LIN {X 0,Y 573.287,Z 367.537,A -85,B 0,C 180,E1 -2259.17,E2 -2259.17} C_VEL
LIN {X 0,Y 573.427,Z 357.093,A -85,B 0,C 180,E1 -2260.058,E2 -2260.058} C_VEL
LIN {X 0,Y 573.544,Z 345.429,A -85,B 0,C 180,E1 -2260.853,E2 -2260.853} C_VEL
LIN {X 0,Y 573.652,Z 334.306,A -85,B 0,C 180,E1 -2261.446,E2 -2261.446} C_VEL
LIN {X 0,Y 573.759,Z 321.162,A -85,B 0,C 180,E1 -2261.974,E2 -2261.974} C_VEL
LIN {X 0,Y 573.832,Z 308.508,A -85,B 0,C 180,E1 -2262.332,E2 -2262.332} C_VEL
LIN {X 0,Y 573.943,Z 295.291,A -85,B 0,C 180,E1 -2262.554,E2 -2262.554} C_VEL
LIN {X 0,Y 573.968,Z 198.701,A -85,B 0,C 180,E1 -2263.769,E2 -2263.769} C_VEL
LIN {X 0,Y 573.396,Z 194.611,A -85,B 0,C 180,E1 -2263.851,E2 -2263.851} C_VEL
LIN {X 0,Y 573.568,Z 174.151,A -85,B 0,C 180,E1 -2266.723,E2 -2266.723} C_VEL
LIN {X 0,Y 573.787,Z 153.426,A -85,B 0,C 180,E1 -2269.647,E2 -2269.647} C_VEL
LIN {X 0,Y 573.932,Z 133.422,A -85,B 0,C 180,E1 -2272.499,E2 -2272.499} C_VEL
LIN {X 0,Y 573.536,Z 128.596,A -85,B 0,C 180,E1 -2273.214,E2 -2273.214} C_VEL
LIN {X 0,Y 573.23,Z 127.084,A -85,B 0,C 180,E1 -2273.466,E2 -2273.466} C_VEL
LIN {X 0,Y 573.214,Z 127.08,A -85,B 0,C 180,E1 -2276.487,E2 -2276.487} C_VEL
LIN {X 0,Y 573.242,Z 127.079,A -85,B 0,C 180,E1 -2279.367,E2 -2279.367} C_VEL
LIN {X 0,Y 573.24,Z 127.076,A -85,B 0,C 180,E1 -2282.226,E2 -2282.226} C_VEL
LIN {X 0,Y 573.225,Z 127.076,A -85,B 0,C 180,E1 -2284.769,E2 -2284.769} C_VEL
LIN {X 0,Y 573.23,Z 127.08,A -85,B 0,C 180,E1 -2287.808,E2 -2287.808} C_VEL
LIN {X 0,Y 573.25,Z 127.073,A -85,B 0,C 180,E1 -2290.525,E2 -2290.525} C_VEL
LIN {X 0,Y 573.21,Z 127.083,A -85,B 0,C 180,E1 -2293.665,E2 -2293.665} C_VEL
LIN {X 0,Y 573.205,Z 127.08,A -85,B 0,C 180,E1 -2296.637,E2 -2296.637} C_VEL
LIN {X 0,Y 573.251,Z 127.078,A -85,B 0,C 180,E1 -2299.475,E2 -2299.475} C_VEL
LIN {X 0,Y 573.23,Z 127.075,A -85,B 0,C 180,E1 -2302.192,E2 -2302.192} C_VEL
LIN {X 0,Y 573.227,Z 127.083,A -85,B 0,C 180,E1 -2305.231,E2 -2305.231} C_VEL
LIN {X 0,Y 573.242,Z 127.074,A -85,B 0,C 180,E1 -2307.774,E2 -2307.774} C_VEL
LIN {X 0,Y 573.236,Z 127.08,A -85,B 0,C 180,E1 -2310.632,E2 -2310.632} C_VEL
LIN {X 0,Y 573.217,Z 127.078,A -85,B 0,C 180,E1 -2313.513,E2 -2313.513} C_VEL
LIN {X 0,Y 573.197,Z 127.081,A -85,B 0,C 180,E1 -2316.133,E2 -2316.133} C_VEL
LIN {X 0,Y 573.232,Z 127.078,A -85,B 0,C 180,E1 -2319.172,E2 -2319.172} C_VEL
LIN {X 0,Y 573.199,Z 127.08,A -85,B 0,C 180,E1 -2321.41,E2 -2321.41} C_VEL
LIN {X 0,Y 573.208,Z 127.084,A -85,B 0,C 180,E1 -2324.351,E2 -2324.351} C_VEL
LIN {X 0,Y 573.196,Z 127.089,A -85,B 0,C 180,E1 -2326.528,E2 -2326.528} C_VEL
LIN {X 0,Y 573.261,Z 127.071,A -85,B 0,C 180,E1 -2329.403,E2 -2329.403} C_VEL
LIN {X 0,Y 573.245,Z 127.081,A -85,B 0,C 180,E1 -2332.249,E2 -2332.249} C_VEL
LIN {X 0,Y 573.279,Z 127.07,A -85,B 0,C 180,E1 -2335.077,E2 -2335.077} C_VEL
LIN {X 0,Y 573.31,Z 127.069,A -85,B 0,C 180,E1 -2337.892,E2 -2337.892} C_VEL
LIN {X 0,Y 573.32,Z 127.07,A -85,B 0,C 180,E1 -2339.999,E2 -2339.999} C_VEL
LIN {X 0,Y 573.277,Z 127.071,A -85,B 0,C 180,E1 -2342.81,E2 -2342.81} C_VEL
LIN {X 0,Y 573.269,Z 127.073,A -85,B 0,C 180,E1 -2345.628,E2 -2345.628} C_VEL
LIN {X 0,Y 573.238,Z 127.078,A -85,B 0,C 180,E1 -2348.46,E2 -2348.46} C_VEL
LIN {X 0,Y 573.239,Z 127.076,A -85,B 0,C 180,E1 -2351.312,E2 -2351.312} C_VEL
LIN {X 0,Y 573.245,Z 127.076,A -85,B 0,C 180,E1 -2354.408,E2 -2354.408} C_VEL
LIN {X 0,Y 573.178,Z 127.083,A -85,B 0,C 180,E1 -2357.113,E2 -2357.113} C_VEL
LIN {X 0,Y 573.206,Z 127.083,A -85,B 0,C 180,E1 -2360.078,E2 -2360.078} C_VEL
LIN {X 0,Y 573.197,Z 127.081,A -85,B 0,C 180,E1 -2362.339,E2 -2362.339} C_VEL
LIN {X 0,Y 573.195,Z 127.081,A -85,B 0,C 180,E1 -2364.348,E2 -2364.348} C_VEL
LIN {X 0,Y 572.558,Z 127.161,A -85,B 0,C 180,E1 -2364.934,E2 -2364.934} C_VEL
LIN {X 0,Y 569.726,Z 127.518,A -85,B 0,C 180,E1 -2365.886,E2 -2365.886} C_VEL
LIN {X 0,Y 567.304,Z 127.823,A -85,B 0,C 180,E1 -2366.652,E2 -2366.652} C_VEL
LIN {X 0,Y 566.246,Z 127.952,A -85,B 0,C 180,E1 -2367.243,E2 -2367.243} C_VEL
LIN {X 0,Y 566.151,Z 127.962,A -85,B 0,C 180,E1 -2367.443,E2 -2367.443} C_VEL
LIN {X 0,Y 566.148,Z 127.963,A -85,B 0,C 180,E1 -2369.771,E2 -2369.771} C_VEL
LIN {X 0,Y 566.19,Z 127.952,A -85,B 0,C 180,E1 -2372.427,E2 -2372.427} C_VEL
LIN {X 0,Y 566.162,Z 127.96,A -85,B 0,C 180,E1 -2374.986,E2 -2374.986} C_VEL
LIN {X 0,Y 566.186,Z 127.96,A -85,B 0,C 180,E1 -2377.461,E2 -2377.461} C_VEL
LIN {X 0,Y 566.192,Z 127.952,A -85,B 0,C 180,E1 -2380.199,E2 -2380.199} C_VEL
LIN {X 0,Y 566.174,Z 127.962,A -85,B 0,C 180,E1 -2383.056,E2 -2383.056} C_VEL
LIN {X 0,Y 566.152,Z 127.957,A -85,B 0,C 180,E1 -2386.053,E2 -2386.053} C_VEL
LIN {X 0,Y 566.15,Z 127.964,A -85,B 0,C 180,E1 -2388.858,E2 -2388.858} C_VEL
LIN {X 0,Y 566.197,Z 127.954,A -85,B 0,C 180,E1 -2391.442,E2 -2391.442} C_VEL
LIN {X 0,Y 566.134,Z 127.961,A -85,B 0,C 180,E1 -2394.305,E2 -2394.305} C_VEL
LIN {X 0,Y 566.187,Z 127.962,A -85,B 0,C 180,E1 -2396.895,E2 -2396.895} C_VEL
LIN {X 0,Y 566.152,Z 127.959,A -85,B 0,C 180,E1 -2399.405,E2 -2399.405} C_VEL
LIN {X 0,Y 566.141,Z 127.959,A -85,B 0,C 180,E1 -2401.853,E2 -2401.853} C_VEL
LIN {X 0,Y 566.18,Z 127.957,A -85,B 0,C 180,E1 -2404.249,E2 -2404.249} C_VEL
LIN {X 0,Y 566.149,Z 127.966,A -85,B 0,C 180,E1 -2406.722,E2 -2406.722} C_VEL
LIN {X 0,Y 566.182,Z 127.958,A -85,B 0,C 180,E1 -2408.901,E2 -2408.901} C_VEL
LIN {X 0,Y 566.175,Z 127.955,A -85,B 0,C 180,E1 -2411.171,E2 -2411.171} C_VEL
LIN {X 0,Y 566.16,Z 127.961,A -85,B 0,C 180,E1 -2414.151,E2 -2414.151} C_VEL
LIN {X 0,Y 566.154,Z 127.967,A -85,B 0,C 180,E1 -2416.358,E2 -2416.358} C_VEL
LIN {X 0,Y 566.202,Z 127.951,A -85,B 0,C 180,E1 -2419.269,E2 -2419.269} C_VEL
LIN {X 0,Y 566.18,Z 127.962,A -85,B 0,C 180,E1 -2422.152,E2 -2422.152} C_VEL
LIN {X 0,Y 566.242,Z 127.946,A -85,B 0,C 180,E1 -2425.016,E2 -2425.016} C_VEL
LIN {X 0,Y 566.272,Z 127.949,A -85,B 0,C 180,E1 -2427.866,E2 -2427.866} C_VEL
LIN {X 0,Y 566.278,Z 127.951,A -85,B 0,C 180,E1 -2430,E2 -2430} C_VEL
LIN {X 0,Y 566.205,Z 127.956,A -85,B 0,C 180,E1 -2432.846,E2 -2432.846} C_VEL
LIN {X 0,Y 566.349,Z 135.714,A -85,B 0,C 180,E1 -2434.27,E2 -2434.27} C_VEL
LIN {X 0,Y 566.262,Z 151.375,A -85,B 0,C 180,E1 -2437.129,E2 -2437.129} C_VEL
LIN {X 0,Y 566.198,Z 156.361,A -85,B 0,C 180,E1 -2438.042,E2 -2438.042} C_VEL
LIN {X 0,Y 567.178,Z 163.364,A -85,B 0,C 180,E1 -2438.167,E2 -2438.167} C_VEL
LIN {X 0,Y 566.934,Z 263.26,A -85,B 0,C 180,E1 -2439.454,E2 -2439.454} C_VEL
LIN {X 0,Y 566.794,Z 276.501,A -85,B 0,C 180,E1 -2439.771,E2 -2439.771} C_VEL
LIN {X 0,Y 566.723,Z 289.134,A -85,B 0,C 180,E1 -2440.224,E2 -2440.224} C_VEL
LIN {X 0,Y 566.591,Z 301.012,A -85,B 0,C 180,E1 -2440.801,E2 -2440.801} C_VEL
LIN {X 0,Y 566.411,Z 312.795,A -85,B 0,C 180,E1 -2441.541,E2 -2441.541} C_VEL
LIN {X 0,Y 566.309,Z 323.203,A -85,B 0,C 180,E1 -2442.361,E2 -2442.361} C_VEL
LIN {X 0,Y 566.179,Z 332.58,A -85,B 0,C 180,E1 -2443.276,E2 -2443.276} C_VEL
LIN {X 0,Y 566.081,Z 341.702,A -85,B 0,C 180,E1 -2444.377,E2 -2444.377} C_VEL
LIN {X 0,Y 566.009,Z 349.047,A -85,B 0,C 180,E1 -2445.483,E2 -2445.483} C_VEL
LIN {X 0,Y 565.939,Z 354.891,A -85,B 0,C 180,E1 -2446.596,E2 -2446.596} C_VEL
LIN {X 0,Y 565.918,Z 359.474,A -85,B 0,C 180,E1 -2447.714,E2 -2447.714} C_VEL
LIN {X 0,Y 565.872,Z 362.921,A -85,B 0,C 180,E1 -2448.839,E2 -2448.839} C_VEL
LIN {X 0,Y 565.841,Z 364.625,A -85,B 0,C 180,E1 -2449.594,E2 -2449.594} C_VEL
LIN {X 0,Y 565.856,Z 365.877,A -85,B 0,C 180,E1 -2450.351,E2 -2450.351} C_VEL
LIN {X 0,Y 565.87,Z 366.787,A -85,B 0,C 180,E1 -2451.335,E2 -2451.335} C_VEL
LIN {X 0,Y 565.838,Z 366.857,A -85,B 0,C 180,E1 -2452.646,E2 -2452.646} C_VEL
LIN {X 0,Y 565.844,Z 366.239,A -85,B 0,C 180,E1 -2453.419,E2 -2453.419} C_VEL
LIN {X 0,Y 565.828,Z 365.168,A -85,B 0,C 180,E1 -2454.198,E2 -2454.198} C_VEL
LIN {X 0,Y 565.908,Z 362.621,A -85,B 0,C 180,E1 -2455.37,E2 -2455.37} C_VEL
LIN {X 0,Y 565.965,Z 358.622,A -85,B 0,C 180,E1 -2456.612,E2 -2456.612} C_VEL
LIN {X 0,Y 565.944,Z 352.622,A -85,B 0,C 180,E1 -2457.956,E2 -2457.956} C_VEL
LIN {X 0,Y 566,Z 345.537,A -85,B 0,C 180,E1 -2459.168,E2 -2459.168} C_VEL
LIN {X 0,Y 566.115,Z 338.044,A -85,B 0,C 180,E1 -2460.184,E2 -2460.184} C_VEL
LIN {X 0,Y 566.242,Z 328.88,A -85,B 0,C 180,E1 -2461.196,E2 -2461.196} C_VEL
LIN {X 0,Y 566.325,Z 319.512,A -85,B 0,C 180,E1 -2462.041,E2 -2462.041} C_VEL
LIN {X 0,Y 566.452,Z 308.728,A -85,B 0,C 180,E1 -2462.826,E2 -2462.826} C_VEL
LIN {X 0,Y 566.637,Z 297.004,A -85,B 0,C 180,E1 -2463.5,E2 -2463.5} C_VEL
LIN {X 0,Y 566.77,Z 285.172,A -85,B 0,C 180,E1 -2464.025,E2 -2464.025} C_VEL
LIN {X 0,Y 566.859,Z 272.362,A -85,B 0,C 180,E1 -2464.435,E2 -2464.435} C_VEL
LIN {X 0,Y 566.968,Z 259.454,A -85,B 0,C 180,E1 -2464.697,E2 -2464.697} C_VEL
LIN {X 0,Y 567.051,Z 161.186,A -85,B 0,C 180,E1 -2465.954,E2 -2465.954} C_VEL
LIN {X 0,Y 566.24,Z 156.369,A -85,B 0,C 180,E1 -2466.045,E2 -2466.045} C_VEL
LIN {X 0,Y 566.424,Z 140.855,A -85,B 0,C 180,E1 -2468.883,E2 -2468.883} C_VEL
LIN {X 0,Y 566.44,Z 130.03,A -85,B 0,C 180,E1 -2470.814,E2 -2470.814} C_VEL
LIN {X 0,Y 566.25,Z 127.951,A -85,B 0,C 180,E1 -2471.222,E2 -2471.222} C_VEL
LIN {X 0,Y 566.197,Z 127.961,A -85,B 0,C 180,E1 -2474.036,E2 -2474.036} C_VEL
LIN {X 0,Y 566.202,Z 127.952,A -85,B 0,C 180,E1 -2477.083,E2 -2477.083} C_VEL
LIN {X 0,Y 566.224,Z 127.959,A -85,B 0,C 180,E1 -2479.803,E2 -2479.803} C_VEL
LIN {X 0,Y 566.196,Z 127.953,A -85,B 0,C 180,E1 -2482.6,E2 -2482.6} C_VEL
LIN {X 0,Y 566.197,Z 127.956,A -85,B 0,C 180,E1 -2485.182,E2 -2485.182} C_VEL
LIN {X 0,Y 566.23,Z 127.954,A -85,B 0,C 180,E1 -2487.744,E2 -2487.744} C_VEL
LIN {X 0,Y 566.202,Z 127.951,A -85,B 0,C 180,E1 -2490.329,E2 -2490.329} C_VEL
LIN {X 0,Y 566.211,Z 127.951,A -85,B 0,C 180,E1 -2492.662,E2 -2492.662} C_VEL
LIN {X 0,Y 566.236,Z 127.953,A -85,B 0,C 180,E1 -2495.04,E2 -2495.04} C_VEL
LIN {X 0,Y 566.193,Z 127.953,A -85,B 0,C 180,E1 -2498.138,E2 -2498.138} C_VEL
LIN {X 0,Y 566.231,Z 127.951,A -85,B 0,C 180,E1 -2500.615,E2 -2500.615} C_VEL
LIN {X 0,Y 566.201,Z 127.955,A -85,B 0,C 180,E1 -2503.413,E2 -2503.413} C_VEL
LIN {X 0,Y 566.186,Z 127.955,A -85,B 0,C 180,E1 -2506.359,E2 -2506.359} C_VEL
LIN {X 0,Y 566.237,Z 127.954,A -85,B 0,C 180,E1 -2508.676,E2 -2508.676} C_VEL
LIN {X 0,Y 566.205,Z 127.951,A -85,B 0,C 180,E1 -2511.435,E2 -2511.435} C_VEL
LIN {X 0,Y 566.263,Z 127.948,A -85,B 0,C 180,E1 -2514.302,E2 -2514.302} C_VEL
LIN {X 0,Y 566.282,Z 127.942,A -85,B 0,C 180,E1 -2517.867,E2 -2517.867} C_VEL
LIN {X 0,Y 566.297,Z 127.943,A -85,B 0,C 180,E1 -2520.712,E2 -2520.712} C_VEL
LIN {X 0,Y 566.255,Z 127.946,A -85,B 0,C 180,E1 -2522.846,E2 -2522.846} C_VEL
LIN {X 0,Y 566.25,Z 127.945,A -85,B 0,C 180,E1 -2525.699,E2 -2525.699} C_VEL
LIN {X 0,Y 566.2,Z 127.954,A -85,B 0,C 180,E1 -2528.567,E2 -2528.567} C_VEL
LIN {X 0,Y 566.243,Z 127.945,A -85,B 0,C 180,E1 -2531.455,E2 -2531.455} C_VEL
LIN {X 0,Y 566.222,Z 127.95,A -85,B 0,C 180,E1 -2534.5,E2 -2534.5} C_VEL
LIN {X 0,Y 566.154,Z 127.958,A -85,B 0,C 180,E1 -2537.334,E2 -2537.334} C_VEL
LIN {X 0,Y 566.194,Z 127.959,A -85,B 0,C 180,E1 -2539.582,E2 -2539.582} C_VEL
LIN {X 0,Y 566.15,Z 127.964,A -85,B 0,C 180,E1 -2541.865,E2 -2541.865} C_VEL
LIN {X 0,Y 566.182,Z 127.956,A -85,B 0,C 180,E1 -2545.021,E2 -2545.021} C_VEL
LIN {X 0,Y 566.16,Z 127.962,A -85,B 0,C 180,E1 -2547.342,E2 -2547.342} C_VEL
LIN {X 0,Y 566.148,Z 127.961,A -85,B 0,C 180,E1 -2549.772,E2 -2549.772} C_VEL
LIN {X 0,Y 566.173,Z 127.955,A -85,B 0,C 180,E1 -2552.425,E2 -2552.425} C_VEL
LIN {X 0,Y 566.152,Z 127.962,A -85,B 0,C 180,E1 -2554.985,E2 -2554.985} C_VEL
LIN {X 0,Y 566.178,Z 127.959,A -85,B 0,C 180,E1 -2557.463,E2 -2557.463} C_VEL
LIN {X 0,Y 566.162,Z 127.957,A -85,B 0,C 180,E1 -2560.203,E2 -2560.203} C_VEL
LIN {X 0,Y 566.148,Z 127.967,A -85,B 0,C 180,E1 -2563.06,E2 -2563.06} C_VEL
LIN {X 0,Y 566.157,Z 127.958,A -85,B 0,C 180,E1 -2566.054,E2 -2566.054} C_VEL
LIN {X 0,Y 566.163,Z 127.96,A -85,B 0,C 180,E1 -2569.22,E2 -2569.22} C_VEL
LIN {X 0,Y 566.173,Z 127.955,A -85,B 0,C 180,E1 -2571.636,E2 -2571.636} C_VEL
LIN {X 0,Y 566.141,Z 127.963,A -85,B 0,C 180,E1 -2574.306,E2 -2574.306} C_VEL
LIN {X 0,Y 566.196,Z 127.956,A -85,B 0,C 180,E1 -2576.896,E2 -2576.896} C_VEL
LIN {X 0,Y 566.169,Z 127.956,A -85,B 0,C 180,E1 -2579.406,E2 -2579.406} C_VEL
LIN {X 0,Y 566.151,Z 127.961,A -85,B 0,C 180,E1 -2581.854,E2 -2581.854} C_VEL
LIN {X 0,Y 566.194,Z 127.962,A -85,B 0,C 180,E1 -2584.25,E2 -2584.25} C_VEL
LIN {X 0,Y 566.203,Z 128.046,A -85,B 0,C 180,E1 -2586.451,E2 -2586.451} C_VEL
LIN {X 0,Y 566.985,Z 133.041,A -85,B 0,C 180,E1 -2587.21,E2 -2587.21} C_VEL
LIN {X 0,Y 566.812,Z 152.847,A -85,B 0,C 180,E1 -2590.064,E2 -2590.064} C_VEL
LIN {X 0,Y 566.588,Z 174.329,A -85,B 0,C 180,E1 -2593.112,E2 -2593.112} C_VEL
LIN {X 0,Y 566.39,Z 194.613,A -85,B 0,C 180,E1 -2595.975,E2 -2595.975} C_VEL
LIN {X 0,Y 567.155,Z 200.513,A -85,B 0,C 180,E1 -2596.085,E2 -2596.085} C_VEL
LIN {X 0,Y 566.961,Z 302.95,A -85,B 0,C 180,E1 -2597.403,E2 -2597.403} C_VEL
LIN {X 0,Y 566.84,Z 316.22,A -85,B 0,C 180,E1 -2597.719,E2 -2597.719} C_VEL
LIN {X 0,Y 566.743,Z 328.379,A -85,B 0,C 180,E1 -2598.148,E2 -2598.148} C_VEL
LIN {X 0,Y 566.604,Z 340.241,A -85,B 0,C 180,E1 -2598.713,E2 -2598.713} C_VEL
LIN {X 0,Y 566.439,Z 352.197,A -85,B 0,C 180,E1 -2599.455,E2 -2599.455} C_VEL
LIN {X 0,Y 566.325,Z 362.605,A -85,B 0,C 180,E1 -2600.266,E2 -2600.266} C_VEL
LIN {X 0,Y 566.207,Z 371.114,A -85,B 0,C 180,E1 -2601.074,E2 -2601.074} C_VEL
LIN {X 0,Y 566.112,Z 378.961,A -85,B 0,C 180,E1 -2601.972,E2 -2601.972} C_VEL
LIN {X 0,Y 566.004,Z 386.623,A -85,B 0,C 180,E1 -2603.047,E2 -2603.047} C_VEL
LIN {X 0,Y 566.004,Z 393.68,A -85,B 0,C 180,E1 -2604.299,E2 -2604.299} C_VEL
LIN {X 0,Y 565.933,Z 398.373,A -85,B 0,C 180,E1 -2605.37,E2 -2605.37} C_VEL
LIN {X 0,Y 565.927,Z 401.958,A -85,B 0,C 180,E1 -2606.44,E2 -2606.44} C_VEL
LIN {X 0,Y 565.878,Z 403.808,A -85,B 0,C 180,E1 -2607.153,E2 -2607.153} C_VEL
LIN {X 0,Y 565.846,Z 406.184,A -85,B 0,C 180,E1 -2608.577,E2 -2608.577} C_VEL
LIN {X 0,Y 565.839,Z 407,A -85,B 0,C 180,E1 -2610,E2 -2610} C_VEL
LIN {X 0,Y 565.846,Z 406.185,A -85,B 0,C 180,E1 -2611.424,E2 -2611.424} C_VEL
LIN {X 0,Y 565.878,Z 403.81,A -85,B 0,C 180,E1 -2612.848,E2 -2612.848} C_VEL
LIN {X 0,Y 565.926,Z 400.895,A -85,B 0,C 180,E1 -2613.917,E2 -2613.917} C_VEL
LIN {X 0,Y 565.878,Z 396.948,A -85,B 0,C 180,E1 -2614.988,E2 -2614.988} C_VEL
LIN {X 0,Y 566.002,Z 391.866,A -85,B 0,C 180,E1 -2616.059,E2 -2616.059} C_VEL
LIN {X 0,Y 566.041,Z 385.466,A -85,B 0,C 180,E1 -2617.132,E2 -2617.132} C_VEL
LIN {X 0,Y 566.134,Z 377.476,A -85,B 0,C 180,E1 -2618.208,E2 -2618.208} C_VEL
LIN {X 0,Y 566.229,Z 369.332,A -85,B 0,C 180,E1 -2619.106,E2 -2619.106} C_VEL
LIN {X 0,Y 566.348,Z 359.396,A -85,B 0,C 180,E1 -2620.005,E2 -2620.005} C_VEL
LIN {X 0,Y 566.536,Z 348.287,A -85,B 0,C 180,E1 -2620.807,E2 -2620.807} C_VEL
LIN {X 0,Y 566.614,Z 337.168,A -85,B 0,C 180,E1 -2621.447,E2 -2621.447} C_VEL
LIN {X 0,Y 566.746,Z 324.973,A -85,B 0,C 180,E1 -2621.988,E2 -2621.988} C_VEL
LIN {X 0,Y 566.914,Z 312.165,A -85,B 0,C 180,E1 -2622.394,E2 -2622.394} C_VEL
LIN {X 0,Y 566.991,Z 300.089,A -85,B 0,C 180,E1 -2622.642,E2 -2622.642} C_VEL
LIN {X 0,Y 567.089,Z 199.595,A -85,B 0,C 180,E1 -2623.928,E2 -2623.928} C_VEL
LIN {X 0,Y 566.392,Z 194.611,A -85,B 0,C 180,E1 -2624.026,E2 -2624.026} C_VEL
LIN {X 0,Y 566.589,Z 174.348,A -85,B 0,C 180,E1 -2626.889,E2 -2626.889} C_VEL
LIN {X 0,Y 566.864,Z 151.61,A -85,B 0,C 180,E1 -2630.124,E2 -2630.124} C_VEL
LIN {X 0,Y 567.001,Z 133.194,A -85,B 0,C 180,E1 -2632.79,E2 -2632.79} C_VEL
LIN {X 0,Y 566.198,Z 127.96,A -85,B 0,C 180,E1 -2633.598,E2 -2633.598} C_VEL
LIN {X 0,Y 566.19,Z 127.955,A -85,B 0,C 180,E1 -2636.543,E2 -2636.543} C_VEL
LIN {X 0,Y 566.173,Z 127.964,A -85,B 0,C 180,E1 -2639.771,E2 -2639.771} C_VEL
LIN {X 0,Y 566.196,Z 127.952,A -85,B 0,C 180,E1 -2642.428,E2 -2642.428} C_VEL
LIN {X 0,Y 566.17,Z 127.957,A -85,B 0,C 180,E1 -2644.987,E2 -2644.987} C_VEL
LIN {X 0,Y 566.194,Z 127.961,A -85,B 0,C 180,E1 -2647.461,E2 -2647.461} C_VEL
LIN {X 0,Y 566.209,Z 127.95,A -85,B 0,C 180,E1 -2650.199,E2 -2650.199} C_VEL
LIN {X 0,Y 566.183,Z 127.958,A -85,B 0,C 180,E1 -2653.056,E2 -2653.056} C_VEL
LIN {X 0,Y 566.16,Z 127.957,A -85,B 0,C 180,E1 -2656.053,E2 -2656.053} C_VEL
LIN {X 0,Y 566.168,Z 127.959,A -85,B 0,C 180,E1 -2658.859,E2 -2658.859} C_VEL
LIN {X 0,Y 566.207,Z 127.955,A -85,B 0,C 180,E1 -2661.443,E2 -2661.443} C_VEL
LIN {X 0,Y 566.146,Z 127.958,A -85,B 0,C 180,E1 -2664.306,E2 -2664.306} C_VEL
LIN {X 0,Y 566.199,Z 127.959,A -85,B 0,C 180,E1 -2666.896,E2 -2666.896} C_VEL
LIN {X 0,Y 566.164,Z 127.959,A -85,B 0,C 180,E1 -2669.406,E2 -2669.406} C_VEL
LIN {X 0,Y 566.154,Z 127.957,A -85,B 0,C 180,E1 -2671.854,E2 -2671.854} C_VEL
LIN {X 0,Y 566.192,Z 127.954,A -85,B 0,C 180,E1 -2674.249,E2 -2674.249} C_VEL
LIN {X 0,Y 566.144,Z 127.96,A -85,B 0,C 180,E1 -2677.366,E2 -2677.366} C_VEL
LIN {X 0,Y 566.174,Z 127.954,A -85,B 0,C 180,E1 -2679.661,E2 -2679.661} C_VEL
LIN {X 0,Y 566.169,Z 127.956,A -85,B 0,C 180,E1 -2681.92,E2 -2681.92} C_VEL
LIN {X 0,Y 566.183,Z 127.958,A -85,B 0,C 180,E1 -2684.89,E2 -2684.89} C_VEL
LIN {X 0,Y 566.177,Z 127.955,A -85,B 0,C 180,E1 -2687.817,E2 -2687.817} C_VEL
LIN {X 0,Y 566.17,Z 127.958,A -85,B 0,C 180,E1 -2689.991,E2 -2689.991} C_VEL
LIN {X 0,Y 566.192,Z 127.955,A -85,B 0,C 180,E1 -2692.869,E2 -2692.869} C_VEL
LIN {X 0,Y 566.255,Z 127.945,A -85,B 0,C 180,E1 -2695.015,E2 -2695.015} C_VEL
LIN {X 0,Y 566.28,Z 127.945,A -85,B 0,C 180,E1 -2697.866,E2 -2697.866} C_VEL
LIN {X 0,Y 566.289,Z 127.946,A -85,B 0,C 180,E1 -2699.999,E2 -2699.999} C_VEL
LIN {X 0,Y 566.245,Z 127.946,A -85,B 0,C 180,E1 -2702.845,E2 -2702.845} C_VEL
LIN {X 0,Y 566.238,Z 127.95,A -85,B 0,C 180,E1 -2705.698,E2 -2705.698} C_VEL
LIN {X 0,Y 566.19,Z 127.954,A -85,B 0,C 180,E1 -2708.566,E2 -2708.566} C_VEL
LIN {X 0,Y 566.197,Z 127.954,A -85,B 0,C 180,E1 -2711.455,E2 -2711.455} C_VEL
LIN {X 0,Y 566.206,Z 127.952,A -85,B 0,C 180,E1 -2714.493,E2 -2714.493} C_VEL
LIN {X 0,Y 566.152,Z 127.96,A -85,B 0,C 180,E1 -2717.332,E2 -2717.332} C_VEL
LIN {X 0,Y 566.176,Z 127.961,A -85,B 0,C 180,E1 -2719.581,E2 -2719.581} C_VEL
LIN {X 0,Y 566.149,Z 127.965,A -85,B 0,C 180,E1 -2721.864,E2 -2721.864} C_VEL
LIN {X 0,Y 566.195,Z 127.953,A -85,B 0,C 180,E1 -2724.962,E2 -2724.962} C_VEL
LIN {X 0,Y 566.151,Z 127.962,A -85,B 0,C 180,E1 -2727.443,E2 -2727.443} C_VEL
LIN {X 0,Y 565.456,Z 128.047,A -85,B 0,C 180,E1 -2728.037,E2 -2728.037} C_VEL
LIN {X 0,Y 562.581,Z 128.404,A -85,B 0,C 180,E1 -2729.001,E2 -2729.001} C_VEL
LIN {X 0,Y 560.182,Z 128.706,A -85,B 0,C 180,E1 -2729.776,E2 -2729.776} C_VEL
LIN {X 0,Y 559.172,Z 128.827,A -85,B 0,C 180,E1 -2730.375,E2 -2730.375} C_VEL
LIN {X 0,Y 559.101,Z 128.836,A -85,B 0,C 180,E1 -2730.578,E2 -2730.578} C_VEL
LIN {X 0,Y 559.146,Z 128.831,A -85,B 0,C 180,E1 -2732.715,E2 -2732.715} C_VEL
LIN {X 0,Y 559.113,Z 128.843,A -85,B 0,C 180,E1 -2735.324,E2 -2735.324} C_VEL
LIN {X 0,Y 559.12,Z 128.834,A -85,B 0,C 180,E1 -2738.018,E2 -2738.018} C_VEL
LIN {X 0,Y 559.146,Z 128.831,A -85,B 0,C 180,E1 -2739.939,E2 -2739.939} C_VEL
LIN {X 0,Y 559.12,Z 128.843,A -85,B 0,C 180,E1 -2743.193,E2 -2743.193} C_VEL
LIN {X 0,Y 559.119,Z 128.834,A -85,B 0,C 180,E1 -2745.763,E2 -2745.763} C_VEL
LIN {X 0,Y 559.097,Z 128.836,A -85,B 0,C 180,E1 -2748.223,E2 -2748.223} C_VEL
LIN {X 0,Y 559.164,Z 128.836,A -85,B 0,C 180,E1 -2751.065,E2 -2751.065} C_VEL
LIN {X 0,Y 559.111,Z 128.834,A -85,B 0,C 180,E1 -2753.787,E2 -2753.787} C_VEL
LIN {X 0,Y 559.138,Z 128.834,A -85,B 0,C 180,E1 -2756.423,E2 -2756.423} C_VEL
LIN {X 0,Y 559.135,Z 128.838,A -85,B 0,C 180,E1 -2758.979,E2 -2758.979} C_VEL
LIN {X 0,Y 559.102,Z 128.835,A -85,B 0,C 180,E1 -2761.63,E2 -2761.63} C_VEL
LIN {X 0,Y 559.147,Z 128.83,A -85,B 0,C 180,E1 -2763.901,E2 -2763.901} C_VEL
LIN {X 0,Y 559.097,Z 128.845,A -85,B 0,C 180,E1 -2766.58,E2 -2766.58} C_VEL
LIN {X 0,Y 559.14,Z 128.831,A -85,B 0,C 180,E1 -2769.394,E2 -2769.394} C_VEL
LIN {X 0,Y 559.106,Z 128.835,A -85,B 0,C 180,E1 -2771.684,E2 -2771.684} C_VEL
LIN {X 0,Y 559.119,Z 128.839,A -85,B 0,C 180,E1 -2774.694,E2 -2774.694} C_VEL
LIN {X 0,Y 559.137,Z 128.832,A -85,B 0,C 180,E1 -2777.662,E2 -2777.662} C_VEL
LIN {X 0,Y 559.111,Z 128.837,A -85,B 0,C 180,E1 -2779.864,E2 -2779.864} C_VEL
LIN {X 0,Y 559.14,Z 128.833,A -85,B 0,C 180,E1 -2782.779,E2 -2782.779} C_VEL
LIN {X 0,Y 559.219,Z 128.821,A -85,B 0,C 180,E1 -2784.953,E2 -2784.953} C_VEL
LIN {X 0,Y 559.242,Z 128.824,A -85,B 0,C 180,E1 -2787.839,E2 -2787.839} C_VEL
LIN {X 0,Y 559.246,Z 128.827,A -85,B 0,C 180,E1 -2790,E2 -2790} C_VEL
LIN {X 0,Y 559.207,Z 129.001,A -85,B 0,C 180,E1 -2792.791,E2 -2792.791} C_VEL
LIN {X 0,Y 559.333,Z 137.274,A -85,B 0,C 180,E1 -2794.323,E2 -2794.323} C_VEL
LIN {X 0,Y 559.255,Z 151.379,A -85,B 0,C 180,E1 -2796.901,E2 -2796.901} C_VEL
LIN {X 0,Y 559.205,Z 156.839,A -85,B 0,C 180,E1 -2797.878,E2 -2797.878} C_VEL
LIN {X 0,Y 560.298,Z 163.935,A -85,B 0,C 180,E1 -2797.999,E2 -2797.999} C_VEL
LIN {X 0,Y 560.014,Z 263.48,A -85,B 0,C 180,E1 -2799.298,E2 -2799.298} C_VEL
LIN {X 0,Y 559.859,Z 276.677,A -85,B 0,C 180,E1 -2799.62,E2 -2799.62} C_VEL
LIN {X 0,Y 559.761,Z 289.277,A -85,B 0,C 180,E1 -2800.078,E2 -2800.078} C_VEL
LIN {X 0,Y 559.617,Z 301.305,A -85,B 0,C 180,E1 -2800.675,E2 -2800.675} C_VEL
LIN {X 0,Y 559.421,Z 313.158,A -85,B 0,C 180,E1 -2801.435,E2 -2801.435} C_VEL
LIN {X 0,Y 559.295,Z 323.247,A -85,B 0,C 180,E1 -2802.242,E2 -2802.242} C_VEL
LIN {X 0,Y 559.144,Z 331.785,A -85,B 0,C 180,E1 -2803.076,E2 -2803.076} C_VEL
LIN {X 0,Y 559.032,Z 340.901,A -85,B 0,C 180,E1 -2804.172,E2 -2804.172} C_VEL
LIN {X 0,Y 558.925,Z 348.515,A -85,B 0,C 180,E1 -2805.311,E2 -2805.311} C_VEL
LIN {X 0,Y 558.858,Z 354.488,A -85,B 0,C 180,E1 -2806.436,E2 -2806.436} C_VEL
LIN {X 0,Y 558.83,Z 359.161,A -85,B 0,C 180,E1 -2807.568,E2 -2807.568} C_VEL
LIN {X 0,Y 558.787,Z 362.693,A -85,B 0,C 180,E1 -2808.706,E2 -2808.706} C_VEL
LIN {X 0,Y 558.743,Z 365.151,A -85,B 0,C 180,E1 -2809.853,E2 -2809.853} C_VEL
LIN {X 0,Y 558.761,Z 366.203,A -85,B 0,C 180,E1 -2810.621,E2 -2810.621} C_VEL
LIN {X 0,Y 558.762,Z 366.864,A -85,B 0,C 180,E1 -2811.449,E2 -2811.449} C_VEL
LIN {X 0,Y 558.737,Z 366.979,A -85,B 0,C 180,E1 -2812.17,E2 -2812.17} C_VEL
LIN {X 0,Y 558.754,Z 366.347,A -85,B 0,C 180,E1 -2813.339,E2 -2813.339} C_VEL
LIN {X 0,Y 558.76,Z 364.628,A -85,B 0,C 180,E1 -2814.524,E2 -2814.524} C_VEL
LIN {X 0,Y 558.817,Z 361.768,A -85,B 0,C 180,E1 -2815.715,E2 -2815.715} C_VEL
LIN {X 0,Y 558.841,Z 357.642,A -85,B 0,C 180,E1 -2816.919,E2 -2816.919} C_VEL
LIN {X 0,Y 558.882,Z 352.629,A -85,B 0,C 180,E1 -2818.029,E2 -2818.029} C_VEL
LIN {X 0,Y 558.924,Z 346.173,A -85,B 0,C 180,E1 -2819.16,E2 -2819.16} C_VEL
LIN {X 0,Y 559.053,Z 338.853,A -85,B 0,C 180,E1 -2820.189,E2 -2820.189} C_VEL
LIN {X 0,Y 559.183,Z 330.471,A -85,B 0,C 180,E1 -2821.15,E2 -2821.15} C_VEL
LIN {X 0,Y 559.302,Z 320.695,A -85,B 0,C 180,E1 -2822.066,E2 -2822.066} C_VEL
LIN {X 0,Y 559.446,Z 309.533,A -85,B 0,C 180,E1 -2822.91,E2 -2822.91} C_VEL
LIN {X 0,Y 559.668,Z 297.404,A -85,B 0,C 180,E1 -2823.625,E2 -2823.625} C_VEL
LIN {X 0,Y 559.831,Z 285.108,A -85,B 0,C 180,E1 -2824.181,E2 -2824.181} C_VEL
LIN {X 0,Y 559.935,Z 272.316,A -85,B 0,C 180,E1 -2824.594,E2 -2824.594} C_VEL
LIN {X 0,Y 560.07,Z 259.384,A -85,B 0,C 180,E1 -2824.858,E2 -2824.858} C_VEL
LIN {X 0,Y 560.25,Z 162.516,A -85,B 0,C 180,E1 -2826.111,E2 -2826.111} C_VEL
LIN {X 0,Y 559.214,Z 156.453,A -85,B 0,C 180,E1 -2826.235,E2 -2826.235} C_VEL
LIN {X 0,Y 559.431,Z 141.938,A -85,B 0,C 180,E1 -2828.913,E2 -2828.913} C_VEL
LIN {X 0,Y 559.332,Z 129.96,A -85,B 0,C 180,E1 -2831.072,E2 -2831.072} C_VEL
LIN {X 0,Y 559.196,Z 128.83,A -85,B 0,C 180,E1 -2831.296,E2 -2831.296} C_VEL
LIN {X 0,Y 559.152,Z 128.837,A -85,B 0,C 180,E1 -2834.24,E2 -2834.24} C_VEL
LIN {X 0,Y 559.161,Z 128.83,A -85,B 0,C 180,E1 -2837.258,E2 -2837.258} C_VEL
LIN {X 0,Y 559.183,Z 128.83,A -85,B 0,C 180,E1 -2840.136,E2 -2840.136} C_VEL
LIN {X 0,Y 559.138,Z 128.833,A -85,B 0,C 180,E1 -2842.892,E2 -2842.892} C_VEL
LIN {X 0,Y 559.164,Z 128.831,A -85,B 0,C 180,E1 -2846.052,E2 -2846.052} C_VEL
LIN {X 0,Y 559.154,Z 128.832,A -85,B 0,C 180,E1 -2848.981,E2 -2848.981} C_VEL
LIN {X 0,Y 559.167,Z 128.834,A -85,B 0,C 180,E1 -2851.62,E2 -2851.62} C_VEL
LIN {X 0,Y 559.179,Z 128.829,A -85,B 0,C 180,E1 -2853.904,E2 -2853.904} C_VEL
LIN {X 0,Y 559.141,Z 128.832,A -85,B 0,C 180,E1 -2856.572,E2 -2856.572} C_VEL
LIN {X 0,Y 559.175,Z 128.832,A -85,B 0,C 180,E1 -2859.396,E2 -2859.396} C_VEL
LIN {X 0,Y 559.133,Z 128.833,A -85,B 0,C 180,E1 -2861.686,E2 -2861.686} C_VEL
LIN {X 0,Y 559.156,Z 128.829,A -85,B 0,C 180,E1 -2863.948,E2 -2863.948} C_VEL
LIN {X 0,Y 559.16,Z 128.829,A -85,B 0,C 180,E1 -2866.184,E2 -2866.184} C_VEL
LIN {X 0,Y 559.208,Z 128.828,A -85,B 0,C 180,E1 -2868.605,E2 -2868.605} C_VEL
LIN {X 0,Y 559.169,Z 128.828,A -85,B 0,C 180,E1 -2871.326,E2 -2871.326} C_VEL
LIN {X 0,Y 559.231,Z 128.823,A -85,B 0,C 180,E1 -2874.23,E2 -2874.23} C_VEL
LIN {X 0,Y 559.253,Z 128.817,A -85,B 0,C 180,E1 -2877.84,E2 -2877.84} C_VEL
LIN {X 0,Y 559.268,Z 128.818,A -85,B 0,C 180,E1 -2880.721,E2 -2880.721} C_VEL
LIN {X 0,Y 559.222,Z 128.822,A -85,B 0,C 180,E1 -2882.882,E2 -2882.882} C_VEL
LIN {X 0,Y 559.219,Z 128.822,A -85,B 0,C 180,E1 -2885.771,E2 -2885.771} C_VEL
LIN {X 0,Y 559.165,Z 128.83,A -85,B 0,C 180,E1 -2888.675,E2 -2888.675} C_VEL
LIN {X 0,Y 559.204,Z 128.823,A -85,B 0,C 180,E1 -2891.601,E2 -2891.601} C_VEL
LIN {X 0,Y 559.185,Z 128.826,A -85,B 0,C 180,E1 -2894.588,E2 -2894.588} C_VEL
LIN {X 0,Y 559.112,Z 128.838,A -85,B 0,C 180,E1 -2897.559,E2 -2897.559} C_VEL
LIN {X 0,Y 559.148,Z 128.837,A -85,B 0,C 180,E1 -2899.839,E2 -2899.839} C_VEL
LIN {X 0,Y 559.105,Z 128.838,A -85,B 0,C 180,E1 -2902.155,E2 -2902.155} C_VEL
LIN {X 0,Y 559.142,Z 128.834,A -85,B 0,C 180,E1 -2905.178,E2 -2905.178} C_VEL
LIN {X 0,Y 559.102,Z 128.842,A -85,B 0,C 180,E1 -2907.717,E2 -2907.717} C_VEL
LIN {X 0,Y 559.094,Z 128.836,A -85,B 0,C 180,E1 -2910.187,E2 -2910.187} C_VEL
LIN {X 0,Y 559.135,Z 128.833,A -85,B 0,C 180,E1 -2912.717,E2 -2912.717} C_VEL
LIN {X 0,Y 559.109,Z 128.843,A -85,B 0,C 180,E1 -2915.326,E2 -2915.326} C_VEL
LIN {X 0,Y 559.098,Z 128.836,A -85,B 0,C 180,E1 -2918.021,E2 -2918.021} C_VEL
LIN {X 0,Y 559.099,Z 128.842,A -85,B 0,C 180,E1 -2920.818,E2 -2920.818} C_VEL
LIN {X 0,Y 559.101,Z 128.837,A -85,B 0,C 180,E1 -2923.738,E2 -2923.738} C_VEL
LIN {X 0,Y 559.102,Z 128.838,A -85,B 0,C 180,E1 -2926.262,E2 -2926.262} C_VEL
LIN {X 0,Y 559.116,Z 128.838,A -85,B 0,C 180,E1 -2929.184,E2 -2929.184} C_VEL
LIN {X 0,Y 559.168,Z 128.831,A -85,B 0,C 180,E1 -2931.193,E2 -2931.193} C_VEL
LIN {X 0,Y 559.118,Z 128.833,A -85,B 0,C 180,E1 -2933.788,E2 -2933.788} C_VEL
LIN {X 0,Y 559.147,Z 128.838,A -85,B 0,C 180,E1 -2936.424,E2 -2936.424} C_VEL
LIN {X 0,Y 559.15,Z 128.833,A -85,B 0,C 180,E1 -2938.98,E2 -2938.98} C_VEL
LIN {X 0,Y 559.112,Z 128.836,A -85,B 0,C 180,E1 -2941.63,E2 -2941.63} C_VEL
LIN {X 0,Y 559.159,Z 128.834,A -85,B 0,C 180,E1 -2943.902,E2 -2943.902} C_VEL
LIN {X 0,Y 559.163,Z 128.927,A -85,B 0,C 180,E1 -2946.311,E2 -2946.311} C_VEL
LIN {X 0,Y 560.048,Z 135.399,A -85,B 0,C 180,E1 -2947.302,E2 -2947.302} C_VEL
LIN {X 0,Y 559.797,Z 155.199,A -85,B 0,C 180,E1 -2950.186,E2 -2950.186} C_VEL
LIN {X 0,Y 559.568,Z 174.343,A -85,B 0,C 180,E1 -2952.936,E2 -2952.936} C_VEL
LIN {X 0,Y 559.374,Z 194.472,A -85,B 0,C 180,E1 -2955.795,E2 -2955.795} C_VEL
LIN {X 0,Y 560.255,Z 202.175,A -85,B 0,C 180,E1 -2955.934,E2 -2955.934} C_VEL
LIN {X 0,Y 560.033,Z 302.948,A -85,B 0,C 180,E1 -2957.245,E2 -2957.245} C_VEL
LIN {X 0,Y 559.913,Z 316.219,A -85,B 0,C 180,E1 -2957.564,E2 -2957.564} C_VEL
LIN {X 0,Y 559.792,Z 328.378,A -85,B 0,C 180,E1 -2957.999,E2 -2957.999} C_VEL
LIN {X 0,Y 559.644,Z 340.058,A -85,B 0,C 180,E1 -2958.56,E2 -2958.56} C_VEL
LIN {X 0,Y 559.458,Z 352.194,A -85,B 0,C 180,E1 -2959.322,E2 -2959.322} C_VEL
LIN {X 0,Y 559.305,Z 362.606,A -85,B 0,C 180,E1 -2960.142,E2 -2960.142} C_VEL
LIN {X 0,Y 559.162,Z 371.114,A -85,B 0,C 180,E1 -2960.961,E2 -2960.961} C_VEL
LIN {X 0,Y 559.05,Z 378.961,A -85,B 0,C 180,E1 -2961.87,E2 -2961.87} C_VEL
LIN {X 0,Y 558.944,Z 386.623,A -85,B 0,C 180,E1 -2962.958,E2 -2962.958} C_VEL
LIN {X 0,Y 558.936,Z 393.68,A -85,B 0,C 180,E1 -2964.227,E2 -2964.227} C_VEL
LIN {X 0,Y 558.826,Z 398.373,A -85,B 0,C 180,E1 -2965.311,E2 -2965.311} C_VEL
LIN {X 0,Y 558.836,Z 401.959,A -85,B 0,C 180,E1 -2966.395,E2 -2966.395} C_VEL
LIN {X 0,Y 558.799,Z 403.807,A -85,B 0,C 180,E1 -2967.116,E2 -2967.116} C_VEL
LIN {X 0,Y 558.745,Z 406.183,A -85,B 0,C 180,E1 -2968.559,E2 -2968.559} C_VEL
LIN {X 0,Y 558.74,Z 407,A -85,B 0,C 180,E1 -2970,E2 -2970} C_VEL
LIN {X 0,Y 558.745,Z 406.184,A -85,B 0,C 180,E1 -2971.442,E2 -2971.442} C_VEL
LIN {X 0,Y 558.799,Z 403.81,A -85,B 0,C 180,E1 -2972.884,E2 -2972.884} C_VEL
LIN {X 0,Y 558.844,Z 400.895,A -85,B 0,C 180,E1 -2973.966,E2 -2973.966} C_VEL
LIN {X 0,Y 558.798,Z 396.947,A -85,B 0,C 180,E1 -2975.051,E2 -2975.051} C_VEL
LIN {X 0,Y 558.922,Z 391.866,A -85,B 0,C 180,E1 -2976.136,E2 -2976.136} C_VEL
LIN {X 0,Y 558.978,Z 385.465,A -85,B 0,C 180,E1 -2977.223,E2 -2977.223} C_VEL
LIN {X 0,Y 559.099,Z 377.475,A -85,B 0,C 180,E1 -2978.312,E2 -2978.312} C_VEL
LIN {X 0,Y 559.195,Z 369.331,A -85,B 0,C 180,E1 -2979.221,E2 -2979.221} C_VEL
LIN {X 0,Y 559.358,Z 359.395,A -85,B 0,C 180,E1 -2980.131,E2 -2980.131} C_VEL
LIN {X 0,Y 559.556,Z 348.393,A -85,B 0,C 180,E1 -2980.937,E2 -2980.937} C_VEL
LIN {X 0,Y 559.673,Z 336.452,A -85,B 0,C 180,E1 -2981.628,E2 -2981.628} C_VEL
LIN {X 0,Y 559.822,Z 324.97,A -85,B 0,C 180,E1 -2982.139,E2 -2982.139} C_VEL
LIN {X 0,Y 559.979,Z 312.163,A -85,B 0,C 180,E1 -2982.55,E2 -2982.55} C_VEL
LIN {X 0,Y 560.08,Z 300.084,A -85,B 0,C 180,E1 -2982.801,E2 -2982.801} C_VEL
LIN {X 0,Y 560.201,Z 200.198,A -85,B 0,C 180,E1 -2984.093,E2 -2984.093} C_VEL
LIN {X 0,Y 559.373,Z 194.49,A -85,B 0,C 180,E1 -2984.205,E2 -2984.205} C_VEL
LIN {X 0,Y 559.57,Z 174.375,A -85,B 0,C 180,E1 -2987.069,E2 -2987.069} C_VEL
LIN {X 0,Y 559.888,Z 152.684,A -85,B 0,C 180,E1 -2990.194,E2 -2990.194} C_VEL
LIN {X 0,Y 560.057,Z 134.283,A -85,B 0,C 180,E1 -2992.893,E2 -2992.893} C_VEL
LIN {X 0,Y 559.156,Z 128.836,A -85,B 0,C 180,E1 -2993.766,E2 -2993.766} C_VEL
LIN {X 0,Y 559.127,Z 128.834,A -85,B 0,C 180,E1 -2996.818,E2 -2996.818} C_VEL
LIN {X 0,Y 559.123,Z 128.841,A -85,B 0,C 180,E1 -2999.852,E2 -2999.852} C_VEL
LIN {X 0,Y 559.151,Z 128.829,A -85,B 0,C 180,E1 -3002.716,E2 -3002.716} C_VEL
LIN {X 0,Y 559.121,Z 128.839,A -85,B 0,C 180,E1 -3005.325,E2 -3005.325} C_VEL
LIN {X 0,Y 559.13,Z 128.834,A -85,B 0,C 180,E1 -3008.018,E2 -3008.018} C_VEL
LIN {X 0,Y 559.157,Z 128.83,A -85,B 0,C 180,E1 -3010.813,E2 -3010.813} C_VEL
LIN {X 0,Y 559.111,Z 128.838,A -85,B 0,C 180,E1 -3013.737,E2 -3013.737} C_VEL
LIN {X 0,Y 559.111,Z 128.834,A -85,B 0,C 180,E1 -3016.263,E2 -3016.263} C_VEL
LIN {X 0,Y 559.157,Z 128.838,A -85,B 0,C 180,E1 -3019.187,E2 -3019.187} C_VEL
LIN {X 0,Y 559.131,Z 128.832,A -85,B 0,C 180,E1 -3021.982,E2 -3021.982} C_VEL
LIN {X 0,Y 559.127,Z 128.837,A -85,B 0,C 180,E1 -3024.789,E2 -3024.789} C_VEL
LIN {X 0,Y 559.153,Z 128.833,A -85,B 0,C 180,E1 -3027.366,E2 -3027.366} C_VEL
LIN {X 0,Y 559.114,Z 128.834,A -85,B 0,C 180,E1 -3030.15,E2 -3030.15} C_VEL
LIN {X 0,Y 559.13,Z 128.837,A -85,B 0,C 180,E1 -3033.182,E2 -3033.182} C_VEL
LIN {X 0,Y 559.11,Z 128.835,A -85,B 0,C 180,E1 -3035.492,E2 -3035.492} C_VEL
LIN {X 0,Y 559.164,Z 128.835,A -85,B 0,C 180,E1 -3038.623,E2 -3038.623} C_VEL
LIN {X 0,Y 559.16,Z 128.834,A -85,B 0,C 180,E1 -3040.925,E2 -3040.925} C_VEL
LIN {X 0,Y 559.13,Z 128.833,A -85,B 0,C 180,E1 -3043.946,E2 -3043.946} C_VEL
LIN {X 0,Y 559.139,Z 128.835,A -85,B 0,C 180,E1 -3046.183,E2 -3046.183} C_VEL
LIN {X 0,Y 559.195,Z 128.825,A -85,B 0,C 180,E1 -3049.133,E2 -3049.133} C_VEL
LIN {X 0,Y 559.181,Z 128.83,A -85,B 0,C 180,E1 -3052.053,E2 -3052.053} C_VEL
LIN {X 0,Y 559.232,Z 128.821,A -85,B 0,C 180,E1 -3054.953,E2 -3054.953} C_VEL
LIN {X 0,Y 559.251,Z 128.82,A -85,B 0,C 180,E1 -3057.839,E2 -3057.839} C_VEL
LIN {X 0,Y 559.258,Z 128.822,A -85,B 0,C 180,E1 -3059.999,E2 -3059.999} C_VEL
LIN {X 0,Y 559.213,Z 128.822,A -85,B 0,C 180,E1 -3062.881,E2 -3062.881} C_VEL
LIN {X 0,Y 559.207,Z 128.827,A -85,B 0,C 180,E1 -3065.77,E2 -3065.77} C_VEL
LIN {X 0,Y 559.155,Z 128.83,A -85,B 0,C 180,E1 -3068.674,E2 -3068.674} C_VEL
LIN {X 0,Y 559.159,Z 128.833,A -85,B 0,C 180,E1 -3071.601,E2 -3071.601} C_VEL
LIN {X 0,Y 559.155,Z 128.83,A -85,B 0,C 180,E1 -3074.575,E2 -3074.575} C_VEL
LIN {X 0,Y 559.111,Z 128.84,A -85,B 0,C 180,E1 -3077.558,E2 -3077.558} C_VEL
LIN {X 0,Y 559.139,Z 128.839,A -85,B 0,C 180,E1 -3079.838,E2 -3079.838} C_VEL
LIN {X 0,Y 559.104,Z 128.838,A -85,B 0,C 180,E1 -3082.154,E2 -3082.154} C_VEL
LIN {X 0,Y 559.14,Z 128.834,A -85,B 0,C 180,E1 -3085.177,E2 -3085.177} C_VEL
LIN {X 0,Y 559.101,Z 128.843,A -85,B 0,C 180,E1 -3087.716,E2 -3087.716} C_VEL
LIN {X 0,Y 559.101,Z 128.836,A -85,B 0,C 180,E1 -3090.578,E2 -3090.578} C_VEL
LIN {X 0,Y 558.461,Z 128.922,A -85,B 0,C 180,E1 -3091.18,E2 -3091.18} C_VEL
LIN {X 0,Y 555.612,Z 129.273,A -85,B 0,C 180,E1 -3092.156,E2 -3092.156} C_VEL
LIN {X 0,Y 553.194,Z 129.574,A -85,B 0,C 180,E1 -3092.942,E2 -3092.942} C_VEL
LIN {X 0,Y 552.162,Z 129.707,A -85,B 0,C 180,E1 -3093.549,E2 -3093.549} C_VEL
LIN {X 0,Y 552.083,Z 129.711,A -85,B 0,C 180,E1 -3093.754,E2 -3093.754} C_VEL
LIN {X 0,Y 552.095,Z 129.71,A -85,B 0,C 180,E1 -3096.747,E2 -3096.747} C_VEL
LIN {X 0,Y 552.119,Z 129.711,A -85,B 0,C 180,E1 -3099.527,E2 -3099.527} C_VEL
LIN {X 0,Y 552.08,Z 129.711,A -85,B 0,C 180,E1 -3102.429,E2 -3102.429} C_VEL
LIN {X 0,Y 552.07,Z 129.715,A -85,B 0,C 180,E1 -3105.559,E2 -3105.559} C_VEL
LIN {X 0,Y 552.056,Z 129.715,A -85,B 0,C 180,E1 -3108.548,E2 -3108.548} C_VEL
LIN {X 0,Y 552.107,Z 129.71,A -85,B 0,C 180,E1 -3111.41,E2 -3111.41} C_VEL
LIN {X 0,Y 552.064,Z 129.713,A -85,B 0,C 180,E1 -3114.154,E2 -3114.154} C_VEL
LIN {X 0,Y 552.1,Z 129.712,A -85,B 0,C 180,E1 -3117.155,E2 -3117.155} C_VEL
LIN {X 0,Y 552.071,Z 129.712,A -85,B 0,C 180,E1 -3119.956,E2 -3119.956} C_VEL
LIN {X 0,Y 552.084,Z 129.714,A -85,B 0,C 180,E1 -3123.009,E2 -3123.009} C_VEL
LIN {X 0,Y 552.067,Z 129.713,A -85,B 0,C 180,E1 -3125.96,E2 -3125.96} C_VEL
LIN {X 0,Y 552.088,Z 129.711,A -85,B 0,C 180,E1 -3129.118,E2 -3129.118} C_VEL
LIN {X 0,Y 552.069,Z 129.711,A -85,B 0,C 180,E1 -3131.442,E2 -3131.442} C_VEL
LIN {X 0,Y 552.077,Z 129.719,A -85,B 0,C 180,E1 -3134.494,E2 -3134.494} C_VEL
LIN {X 0,Y 552.09,Z 129.713,A -85,B 0,C 180,E1 -3136.754,E2 -3136.754} C_VEL
LIN {X 0,Y 552.076,Z 129.712,A -85,B 0,C 180,E1 -3139.734,E2 -3139.734} C_VEL
LIN {X 0,Y 552.1,Z 129.712,A -85,B 0,C 180,E1 -3141.95,E2 -3141.95} C_VEL
LIN {X 0,Y 552.196,Z 129.697,A -85,B 0,C 180,E1 -3144.888,E2 -3144.888} C_VEL
LIN {X 0,Y 552.213,Z 129.7,A -85,B 0,C 180,E1 -3147.812,E2 -3147.812} C_VEL
LIN {X 0,Y 552.215,Z 129.703,A -85,B 0,C 180,E1 -3150,E2 -3150} C_VEL
LIN {X 0,Y 552.184,Z 129.852,A -85,B 0,C 180,E1 -3152.69,E2 -3152.69} C_VEL
LIN {X 0,Y 552.336,Z 136.902,A -85,B 0,C 180,E1 -3154.013,E2 -3154.013} C_VEL
LIN {X 0,Y 552.268,Z 151.561,A -85,B 0,C 180,E1 -3156.704,E2 -3156.704} C_VEL
LIN {X 0,Y 552.189,Z 156.754,A -85,B 0,C 180,E1 -3157.678,E2 -3157.678} C_VEL
LIN {X 0,Y 553.42,Z 164.675,A -85,B 0,C 180,E1 -3157.827,E2 -3157.827} C_VEL
LIN {X 0,Y 553.09,Z 263.83,A -85,B 0,C 180,E1 -3159.139,E2 -3159.139} C_VEL
LIN {X 0,Y 552.928,Z 276.991,A -85,B 0,C 180,E1 -3159.465,E2 -3159.465} C_VEL
LIN {X 0,Y 552.816,Z 289.576,A -85,B 0,C 180,E1 -3159.929,E2 -3159.929} C_VEL
LIN {X 0,Y 552.653,Z 301.595,A -85,B 0,C 180,E1 -3160.533,E2 -3160.533} C_VEL
LIN {X 0,Y 552.442,Z 312.709,A -85,B 0,C 180,E1 -3161.251,E2 -3161.251} C_VEL
LIN {X 0,Y 552.301,Z 323.465,A -85,B 0,C 180,E1 -3162.12,E2 -3162.12} C_VEL
LIN {X 0,Y 552.111,Z 332.792,A -85,B 0,C 180,E1 -3163.058,E2 -3163.058} C_VEL
LIN {X 0,Y 551.978,Z 341.565,A -85,B 0,C 180,E1 -3164.148,E2 -3164.148} C_VEL
LIN {X 0,Y 551.857,Z 349.147,A -85,B 0,C 180,E1 -3165.323,E2 -3165.323} C_VEL
LIN {X 0,Y 551.782,Z 354.074,A -85,B 0,C 180,E1 -3166.273,E2 -3166.273} C_VEL
LIN {X 0,Y 551.744,Z 358.972,A -85,B 0,C 180,E1 -3167.455,E2 -3167.455} C_VEL
LIN {X 0,Y 551.697,Z 362.463,A -85,B 0,C 180,E1 -3168.57,E2 -3168.57} C_VEL
LIN {X 0,Y 551.676,Z 364.543,A -85,B 0,C 180,E1 -3169.491,E2 -3169.491} C_VEL
LIN {X 0,Y 551.655,Z 366.511,A -85,B 0,C 180,E1 -3170.899,E2 -3170.899} C_VEL
LIN {X 0,Y 551.645,Z 366.927,A -85,B 0,C 180,E1 -3171.682,E2 -3171.682} C_VEL
LIN {X 0,Y 551.64,Z 366.913,A -85,B 0,C 180,E1 -3172.47,E2 -3172.47} C_VEL
LIN {X 0,Y 551.654,Z 366.218,A -85,B 0,C 180,E1 -3173.472,E2 -3173.472} C_VEL
LIN {X 0,Y 551.682,Z 364.023,A -85,B 0,C 180,E1 -3174.859,E2 -3174.859} C_VEL
LIN {X 0,Y 551.74,Z 360.874,A -85,B 0,C 180,E1 -3176.069,E2 -3176.069} C_VEL
LIN {X 0,Y 551.773,Z 356.401,A -85,B 0,C 180,E1 -3177.293,E2 -3177.293} C_VEL
LIN {X 0,Y 551.829,Z 350.569,A -85,B 0,C 180,E1 -3178.507,E2 -3178.507} C_VEL
LIN {X 0,Y 551.899,Z 344.17,A -85,B 0,C 180,E1 -3179.568,E2 -3179.568} C_VEL
LIN {X 0,Y 552.026,Z 336.4,A -85,B 0,C 180,E1 -3180.614,E2 -3180.614} C_VEL
LIN {X 0,Y 552.213,Z 326.908,A -85,B 0,C 180,E1 -3181.646,E2 -3181.646} C_VEL
LIN {X 0,Y 552.38,Z 316.033,A -85,B 0,C 180,E1 -3182.592,E2 -3182.592} C_VEL
LIN {X 0,Y 552.612,Z 304.789,A -85,B 0,C 180,E1 -3183.37,E2 -3183.37} C_VEL
LIN {X 0,Y 552.782,Z 292.778,A -85,B 0,C 180,E1 -3184.015,E2 -3184.015} C_VEL
LIN {X 0,Y 552.941,Z 280.583,A -85,B 0,C 180,E1 -3184.509,E2 -3184.509} C_VEL
LIN {X 0,Y 553.071,Z 267.441,A -85,B 0,C 180,E1 -3184.878,E2 -3184.878} C_VEL
LIN {X 0,Y 553.131,Z 250.082,A -85,B 0,C 180,E1 -3185.151,E2 -3185.151} C_VEL
LIN {X 0,Y 553.302,Z 162.974,A -85,B 0,C 180,E1 -3186.288,E2 -3186.288} C_VEL
LIN {X 0,Y 552.198,Z 156.677,A -85,B 0,C 180,E1 -3186.405,E2 -3186.405} C_VEL
LIN {X 0,Y 552.432,Z 142.144,A -85,B 0,C 180,E1 -3189.102,E2 -3189.102} C_VEL
LIN {X 0,Y 552.344,Z 131.176,A -85,B 0,C 180,E1 -3191.102,E2 -3191.102} C_VEL
LIN {X 0,Y 552.188,Z 129.704,A -85,B 0,C 180,E1 -3191.396,E2 -3191.396} C_VEL
LIN {X 0,Y 552.093,Z 129.713,A -85,B 0,C 180,E1 -3194.533,E2 -3194.533} C_VEL
LIN {X 0,Y 552.128,Z 129.71,A -85,B 0,C 180,E1 -3197.585,E2 -3197.585} C_VEL
LIN {X 0,Y 552.132,Z 129.706,A -85,B 0,C 180,E1 -3200.474,E2 -3200.474} C_VEL
LIN {X 0,Y 552.104,Z 129.713,A -85,B 0,C 180,E1 -3203.318,E2 -3203.318} C_VEL
LIN {X 0,Y 552.125,Z 129.709,A -85,B 0,C 180,E1 -3205.94,E2 -3205.94} C_VEL
LIN {X 0,Y 552.117,Z 129.706,A -85,B 0,C 180,E1 -3208.541,E2 -3208.541} C_VEL
LIN {X 0,Y 552.123,Z 129.715,A -85,B 0,C 180,E1 -3211.439,E2 -3211.439} C_VEL
LIN {X 0,Y 552.129,Z 129.705,A -85,B 0,C 180,E1 -3214.357,E2 -3214.357} C_VEL
LIN {X 0,Y 552.098,Z 129.711,A -85,B 0,C 180,E1 -3216.759,E2 -3216.759} C_VEL
LIN {X 0,Y 552.118,Z 129.714,A -85,B 0,C 180,E1 -3219.12,E2 -3219.12} C_VEL
LIN {X 0,Y 552.091,Z 129.713,A -85,B 0,C 180,E1 -3221.444,E2 -3221.444} C_VEL
LIN {X 0,Y 552.105,Z 129.708,A -85,B 0,C 180,E1 -3223.738,E2 -3223.738} C_VEL
LIN {X 0,Y 552.123,Z 129.705,A -85,B 0,C 180,E1 -3226.005,E2 -3226.005} C_VEL
LIN {X 0,Y 552.162,Z 129.707,A -85,B 0,C 180,E1 -3228.994,E2 -3228.994} C_VEL
LIN {X 0,Y 552.151,Z 129.701,A -85,B 0,C 180,E1 -3231.952,E2 -3231.952} C_VEL
LIN {X 0,Y 552.222,Z 129.696,A -85,B 0,C 180,E1 -3234.89,E2 -3234.89} C_VEL
LIN {X 0,Y 552.224,Z 129.693,A -85,B 0,C 180,E1 -3237.813,E2 -3237.813} C_VEL
LIN {X 0,Y 552.238,Z 129.693,A -85,B 0,C 180,E1 -3240.73,E2 -3240.73} C_VEL
LIN {X 0,Y 552.188,Z 129.698,A -85,B 0,C 180,E1 -3242.919,E2 -3242.919} C_VEL
LIN {X 0,Y 552.188,Z 129.698,A -85,B 0,C 180,E1 -3245.845,E2 -3245.845} C_VEL
LIN {X 0,Y 552.136,Z 129.704,A -85,B 0,C 180,E1 -3248.787,E2 -3248.787} C_VEL
LIN {X 0,Y 552.16,Z 129.702,A -85,B 0,C 180,E1 -3251.751,E2 -3251.751} C_VEL
LIN {X 0,Y 552.131,Z 129.704,A -85,B 0,C 180,E1 -3254.749,E2 -3254.749} C_VEL
LIN {X 0,Y 552.078,Z 129.718,A -85,B 0,C 180,E1 -3257.79,E2 -3257.79} C_VEL
LIN {X 0,Y 552.1,Z 129.711,A -85,B 0,C 180,E1 -3260.103,E2 -3260.103} C_VEL
LIN {X 0,Y 552.045,Z 129.715,A -85,B 0,C 180,E1 -3262.454,E2 -3262.454} C_VEL
LIN {X 0,Y 552.085,Z 129.715,A -85,B 0,C 180,E1 -3265.334,E2 -3265.334} C_VEL
LIN {X 0,Y 552.05,Z 129.716,A -85,B 0,C 180,E1 -3268.102,E2 -3268.102} C_VEL
LIN {X 0,Y 552.069,Z 129.711,A -85,B 0,C 180,E1 -3270.612,E2 -3270.612} C_VEL
LIN {X 0,Y 552.09,Z 129.717,A -85,B 0,C 180,E1 -3273.188,E2 -3273.188} C_VEL
LIN {X 0,Y 552.064,Z 129.714,A -85,B 0,C 180,E1 -3275.846,E2 -3275.846} C_VEL
LIN {X 0,Y 552.074,Z 129.713,A -85,B 0,C 180,E1 -3278.593,E2 -3278.593} C_VEL
LIN {X 0,Y 552.055,Z 129.718,A -85,B 0,C 180,E1 -3281.453,E2 -3281.453} C_VEL
LIN {X 0,Y 552.076,Z 129.715,A -85,B 0,C 180,E1 -3284.53,E2 -3284.53} C_VEL
LIN {X 0,Y 552.082,Z 129.712,A -85,B 0,C 180,E1 -3287.591,E2 -3287.591} C_VEL
LIN {X 0,Y 552.123,Z 129.712,A -85,B 0,C 180,E1 -3290.472,E2 -3290.472} C_VEL
LIN {X 0,Y 552.099,Z 129.708,A -85,B 0,C 180,E1 -3293.319,E2 -3293.319} C_VEL
LIN {X 0,Y 552.099,Z 129.71,A -85,B 0,C 180,E1 -3295.937,E2 -3295.937} C_VEL
LIN {X 0,Y 552.123,Z 129.714,A -85,B 0,C 180,E1 -3298.541,E2 -3298.541} C_VEL
LIN {X 0,Y 552.081,Z 129.712,A -85,B 0,C 180,E1 -3301.447,E2 -3301.447} C_VEL
LIN {X 0,Y 552.085,Z 129.719,A -85,B 0,C 180,E1 -3304.354,E2 -3304.354} C_VEL
LIN {X 0,Y 552.132,Z 129.908,A -85,B 0,C 180,E1 -3306.183,E2 -3306.183} C_VEL
LIN {X 0,Y 553.094,Z 136.433,A -85,B 0,C 180,E1 -3307.198,E2 -3307.198} C_VEL
LIN {X 0,Y 552.852,Z 154.917,A -85,B 0,C 180,E1 -3309.926,E2 -3309.926} C_VEL
LIN {X 0,Y 552.559,Z 174.836,A -85,B 0,C 180,E1 -3312.824,E2 -3312.824} C_VEL
LIN {X 0,Y 552.362,Z 194.31,A -85,B 0,C 180,E1 -3315.627,E2 -3315.627} C_VEL
LIN {X 0,Y 553.357,Z 202.397,A -85,B 0,C 180,E1 -3315.762,E2 -3315.762} C_VEL
LIN {X 0,Y 553.104,Z 302.624,A -85,B 0,C 180,E1 -3317.082,E2 -3317.082} C_VEL
LIN {X 0,Y 552.98,Z 315.938,A -85,B 0,C 180,E1 -3317.406,E2 -3317.406} C_VEL
LIN {X 0,Y 552.847,Z 328.133,A -85,B 0,C 180,E1 -3317.846,E2 -3317.846} C_VEL
LIN {X 0,Y 552.657,Z 338.966,A -85,B 0,C 180,E1 -3318.365,E2 -3318.365} C_VEL
LIN {X 0,Y 552.482,Z 350.76,A -85,B 0,C 180,E1 -3319.093,E2 -3319.093} C_VEL
LIN {X 0,Y 552.298,Z 361.448,A -85,B 0,C 180,E1 -3319.923,E2 -3319.923} C_VEL
LIN {X 0,Y 552.131,Z 371.079,A -85,B 0,C 180,E1 -3320.845,E2 -3320.845} C_VEL
LIN {X 0,Y 552.013,Z 378.961,A -85,B 0,C 180,E1 -3321.765,E2 -3321.765} C_VEL
LIN {X 0,Y 551.89,Z 386.622,A -85,B 0,C 180,E1 -3322.868,E2 -3322.868} C_VEL
LIN {X 0,Y 551.867,Z 393.68,A -85,B 0,C 180,E1 -3324.153,E2 -3324.153} C_VEL
LIN {X 0,Y 551.725,Z 398.373,A -85,B 0,C 180,E1 -3325.251,E2 -3325.251} C_VEL
LIN {X 0,Y 551.75,Z 401.958,A -85,B 0,C 180,E1 -3326.349,E2 -3326.349} C_VEL
LIN {X 0,Y 551.724,Z 403.807,A -85,B 0,C 180,E1 -3327.079,E2 -3327.079} C_VEL
LIN {X 0,Y 551.645,Z 406.182,A -85,B 0,C 180,E1 -3328.54,E2 -3328.54} C_VEL
LIN {X 0,Y 551.64,Z 407,A -85,B 0,C 180,E1 -3330,E2 -3330} C_VEL
LIN {X 0,Y 551.645,Z 406.183,A -85,B 0,C 180,E1 -3331.46,E2 -3331.46} C_VEL
LIN {X 0,Y 551.724,Z 403.81,A -85,B 0,C 180,E1 -3332.921,E2 -3332.921} C_VEL
LIN {X 0,Y 551.764,Z 400.895,A -85,B 0,C 180,E1 -3334.017,E2 -3334.017} C_VEL
LIN {X 0,Y 551.724,Z 396.947,A -85,B 0,C 180,E1 -3335.116,E2 -3335.116} C_VEL
LIN {X 0,Y 551.825,Z 391.191,A -85,B 0,C 180,E1 -3336.341,E2 -3336.341} C_VEL
LIN {X 0,Y 551.927,Z 384.234,A -85,B 0,C 180,E1 -3337.5,E2 -3337.5} C_VEL
LIN {X 0,Y 552.083,Z 375.985,A -85,B 0,C 180,E1 -3338.603,E2 -3338.603} C_VEL
LIN {X 0,Y 552.201,Z 367.485,A -85,B 0,C 180,E1 -3339.524,E2 -3339.524} C_VEL
LIN {X 0,Y 552.429,Z 356.983,A -85,B 0,C 180,E1 -3340.445,E2 -3340.445} C_VEL
LIN {X 0,Y 552.576,Z 346.127,A -85,B 0,C 180,E1 -3341.214,E2 -3341.214} C_VEL
LIN {X 0,Y 552.753,Z 335.201,A -85,B 0,C 180,E1 -3341.831,E2 -3341.831} C_VEL
LIN {X 0,Y 552.899,Z 323.515,A -85,B 0,C 180,E1 -3342.34,E2 -3342.34} C_VEL
LIN {X 0,Y 553.037,Z 310.966,A -85,B 0,C 180,E1 -3342.733,E2 -3342.733} C_VEL
LIN {X 0,Y 553.204,Z 298.257,A -85,B 0,C 180,E1 -3342.986,E2 -3342.986} C_VEL
LIN {X 0,Y 553.233,Z 200.351,A -85,B 0,C 180,E1 -3344.269,E2 -3344.269} C_VEL
LIN {X 0,Y 552.346,Z 194.229,A -85,B 0,C 180,E1 -3344.393,E2 -3344.393} C_VEL
LIN {X 0,Y 552.583,Z 173.738,A -85,B 0,C 180,E1 -3347.35,E2 -3347.35} C_VEL
LIN {X 0,Y 552.941,Z 152.444,A -85,B 0,C 180,E1 -3350.459,E2 -3350.459} C_VEL
LIN {X 0,Y 553.083,Z 135.372,A -85,B 0,C 180,E1 -3353.001,E2 -3353.001} C_VEL
LIN {X 0,Y 552.085,Z 129.716,A -85,B 0,C 180,E1 -3353.916,E2 -3353.916} C_VEL
LIN {X 0,Y 552.096,Z 129.711,A -85,B 0,C 180,E1 -3356.99,E2 -3356.99} C_VEL
LIN {X 0,Y 552.099,Z 129.713,A -85,B 0,C 180,E1 -3360.047,E2 -3360.047} C_VEL
LIN {X 0,Y 552.111,Z 129.707,A -85,B 0,C 180,E1 -3362.845,E2 -3362.845} C_VEL
LIN {X 0,Y 552.075,Z 129.715,A -85,B 0,C 180,E1 -3365.845,E2 -3365.845} C_VEL
LIN {X 0,Y 552.116,Z 129.706,A -85,B 0,C 180,E1 -3368.59,E2 -3368.59} C_VEL
LIN {X 0,Y 552.078,Z 129.719,A -85,B 0,C 180,E1 -3371.45,E2 -3371.45} C_VEL
LIN {X 0,Y 552.079,Z 129.711,A -85,B 0,C 180,E1 -3374.529,E2 -3374.529} C_VEL
LIN {X 0,Y 552.091,Z 129.713,A -85,B 0,C 180,E1 -3377.59,E2 -3377.59} C_VEL
LIN {X 0,Y 552.13,Z 129.705,A -85,B 0,C 180,E1 -3380.472,E2 -3380.472} C_VEL
LIN {X 0,Y 552.103,Z 129.713,A -85,B 0,C 180,E1 -3383.318,E2 -3383.318} C_VEL
LIN {X 0,Y 552.102,Z 129.707,A -85,B 0,C 180,E1 -3385.937,E2 -3385.937} C_VEL
LIN {X 0,Y 552.084,Z 129.713,A -85,B 0,C 180,E1 -3388.538,E2 -3388.538} C_VEL
LIN {X 0,Y 552.083,Z 129.712,A -85,B 0,C 180,E1 -3391.447,E2 -3391.447} C_VEL
LIN {X 0,Y 552.087,Z 129.712,A -85,B 0,C 180,E1 -3394.353,E2 -3394.353} C_VEL
LIN {X 0,Y 552.072,Z 129.72,A -85,B 0,C 180,E1 -3396.756,E2 -3396.756} C_VEL
LIN {X 0,Y 552.101,Z 129.711,A -85,B 0,C 180,E1 -3399.119,E2 -3399.119} C_VEL
LIN {X 0,Y 552.083,Z 129.71,A -85,B 0,C 180,E1 -3401.442,E2 -3401.442} C_VEL
LIN {X 0,Y 552.09,Z 129.717,A -85,B 0,C 180,E1 -3404.494,E2 -3404.494} C_VEL
LIN {X 0,Y 552.107,Z 129.707,A -85,B 0,C 180,E1 -3407.502,E2 -3407.502} C_VEL
LIN {X 0,Y 552.1,Z 129.708,A -85,B 0,C 180,E1 -3409.734,E2 -3409.734} C_VEL
LIN {X 0,Y 552.139,Z 129.706,A -85,B 0,C 180,E1 -3411.951,E2 -3411.951} C_VEL
LIN {X 0,Y 552.209,Z 129.696,A -85,B 0,C 180,E1 -3414.888,E2 -3414.888} C_VEL
LIN {X 0,Y 552.222,Z 129.695,A -85,B 0,C 180,E1 -3417.811,E2 -3417.811} C_VEL
LIN {X 0,Y 552.226,Z 129.698,A -85,B 0,C 180,E1 -3419.999,E2 -3419.999} C_VEL
LIN {X 0,Y 552.18,Z 129.698,A -85,B 0,C 180,E1 -3422.918,E2 -3422.918} C_VEL
LIN {X 0,Y 552.177,Z 129.704,A -85,B 0,C 180,E1 -3425.843,E2 -3425.843} C_VEL
LIN {X 0,Y 552.127,Z 129.705,A -85,B 0,C 180,E1 -3428.786,E2 -3428.786} C_VEL
LIN {X 0,Y 552.105,Z 129.713,A -85,B 0,C 180,E1 -3431.751,E2 -3431.751} C_VEL
LIN {X 0,Y 552.122,Z 129.705,A -85,B 0,C 180,E1 -3434.748,E2 -3434.748} C_VEL
LIN {X 0,Y 552.075,Z 129.721,A -85,B 0,C 180,E1 -3437.789,E2 -3437.789} C_VEL
LIN {X 0,Y 552.094,Z 129.712,A -85,B 0,C 180,E1 -3440.102,E2 -3440.102} C_VEL
LIN {X 0,Y 552.045,Z 129.715,A -85,B 0,C 180,E1 -3442.452,E2 -3442.452} C_VEL
LIN {X 0,Y 552.083,Z 129.715,A -85,B 0,C 180,E1 -3445.333,E2 -3445.333} C_VEL
LIN {X 0,Y 552.049,Z 129.716,A -85,B 0,C 180,E1 -3448.101,E2 -3448.101} C_VEL
LIN {X 0,Y 552.07,Z 129.711,A -85,B 0,C 180,E1 -3450.61,E2 -3450.61} C_VEL
LIN {X 0,Y 552.102,Z 129.713,A -85,B 0,C 180,E1 -3453.186,E2 -3453.186} C_VEL
LIN {X 0,Y 552.083,Z 129.711,A -85,B 0,C 180,E1 -3453.754,E2 -3453.754} C_VEL
LIN {X 0,Y 551.44,Z 129.793,A -85,B 0,C 180,E1 -3454.363,E2 -3454.363} C_VEL
LIN {X 0,Y 548.629,Z 130.149,A -85,B 0,C 180,E1 -3455.351,E2 -3455.351} C_VEL
LIN {X 0,Y 546.223,Z 130.444,A -85,B 0,C 180,E1 -3456.147,E2 -3456.147} C_VEL
LIN {X 0,Y 545.159,Z 130.574,A -85,B 0,C 180,E1 -3456.761,E2 -3456.761} C_VEL
LIN {X 0,Y 545.056,Z 130.589,A -85,B 0,C 180,E1 -3456.969,E2 -3456.969} C_VEL
LIN {X 0,Y 545.048,Z 130.586,A -85,B 0,C 180,E1 -3460.143,E2 -3460.143} C_VEL
LIN {X 0,Y 545.013,Z 130.599,A -85,B 0,C 180,E1 -3463.112,E2 -3463.112} C_VEL
LIN {X 0,Y 545.023,Z 130.589,A -85,B 0,C 180,E1 -3466.228,E2 -3466.228} C_VEL
LIN {X 0,Y 545.011,Z 130.597,A -85,B 0,C 180,E1 -3468.878,E2 -3468.878} C_VEL
LIN {X 0,Y 545.041,Z 130.587,A -85,B 0,C 180,E1 -3471.761,E2 -3471.761} C_VEL
LIN {X 0,Y 545.018,Z 130.594,A -85,B 0,C 180,E1 -3474.53,E2 -3474.53} C_VEL
LIN {X 0,Y 545.055,Z 130.589,A -85,B 0,C 180,E1 -3477.21,E2 -3477.21} C_VEL
LIN {X 0,Y 545.02,Z 130.59,A -85,B 0,C 180,E1 -3479.807,E2 -3479.807} C_VEL
LIN {X 0,Y 545.027,Z 130.596,A -85,B 0,C 180,E1 -3482.839,E2 -3482.839} C_VEL
LIN {X 0,Y 545.011,Z 130.591,A -85,B 0,C 180,E1 -3485.629,E2 -3485.629} C_VEL
LIN {X 0,Y 545.027,Z 130.594,A -85,B 0,C 180,E1 -3488.835,E2 -3488.835} C_VEL
LIN {X 0,Y 545.033,Z 130.589,A -85,B 0,C 180,E1 -3491.194,E2 -3491.194} C_VEL
LIN {X 0,Y 545.024,Z 130.596,A -85,B 0,C 180,E1 -3494.288,E2 -3494.288} C_VEL
LIN {X 0,Y 545.04,Z 130.593,A -85,B 0,C 180,E1 -3496.579,E2 -3496.579} C_VEL
LIN {X 0,Y 545.063,Z 130.586,A -85,B 0,C 180,E1 -3498.848,E2 -3498.848} C_VEL
LIN {X 0,Y 545.058,Z 130.588,A -85,B 0,C 180,E1 -3501.846,E2 -3501.846} C_VEL
LIN {X 0,Y 545.154,Z 130.574,A -85,B 0,C 180,E1 -3504.822,E2 -3504.822} C_VEL
LIN {X 0,Y 545.183,Z 130.575,A -85,B 0,C 180,E1 -3507.783,E2 -3507.783} C_VEL
LIN {X 0,Y 545.183,Z 130.579,A -85,B 0,C 180,E1 -3510,E2 -3510} C_VEL
LIN {X 0,Y 545.154,Z 130.71,A -85,B 0,C 180,E1 -3512.586,E2 -3512.586} C_VEL
LIN {X 0,Y 545.352,Z 138.532,A -85,B 0,C 180,E1 -3514.064,E2 -3514.064} C_VEL
LIN {X 0,Y 545.241,Z 154.513,A -85,B 0,C 180,E1 -3517.026,E2 -3517.026} C_VEL
LIN {X 0,Y 545.195,Z 157.005,A -85,B 0,C 180,E1 -3517.5,E2 -3517.5} C_VEL
LIN {X 0,Y 546.56,Z 165.33,A -85,B 0,C 180,E1 -3517.651,E2 -3517.651} C_VEL
LIN {X 0,Y 546.185,Z 264.151,A -85,B 0,C 180,E1 -3518.976,E2 -3518.976} C_VEL
LIN {X 0,Y 546.007,Z 277.298,A -85,B 0,C 180,E1 -3519.305,E2 -3519.305} C_VEL
LIN {X 0,Y 545.9,Z 289.85,A -85,B 0,C 180,E1 -3519.775,E2 -3519.775} C_VEL
LIN {X 0,Y 545.694,Z 301.883,A -85,B 0,C 180,E1 -3520.388,E2 -3520.388} C_VEL
LIN {X 0,Y 545.463,Z 313.393,A -85,B 0,C 180,E1 -3521.143,E2 -3521.143} C_VEL
LIN {X 0,Y 545.316,Z 323.738,A -85,B 0,C 180,E1 -3521.994,E2 -3521.994} C_VEL
LIN {X 0,Y 545.111,Z 332.238,A -85,B 0,C 180,E1 -3522.85,E2 -3522.85} C_VEL
LIN {X 0,Y 544.952,Z 341.434,A -85,B 0,C 180,E1 -3523.993,E2 -3523.993} C_VEL
LIN {X 0,Y 544.795,Z 348.867,A -85,B 0,C 180,E1 -3525.143,E2 -3525.143} C_VEL
LIN {X 0,Y 544.721,Z 353.876,A -85,B 0,C 180,E1 -3526.105,E2 -3526.105} C_VEL
LIN {X 0,Y 544.663,Z 358.814,A -85,B 0,C 180,E1 -3527.286,E2 -3527.286} C_VEL
LIN {X 0,Y 544.612,Z 362.425,A -85,B 0,C 180,E1 -3528.431,E2 -3528.431} C_VEL
LIN {X 0,Y 544.573,Z 365.034,A -85,B 0,C 180,E1 -3529.606,E2 -3529.606} C_VEL
LIN {X 0,Y 544.558,Z 366.188,A -85,B 0,C 180,E1 -3530.393,E2 -3530.393} C_VEL
LIN {X 0,Y 544.563,Z 367.115,A -85,B 0,C 180,E1 -3531.69,E2 -3531.69} C_VEL
LIN {X 0,Y 544.542,Z 366.976,A -85,B 0,C 180,E1 -3532.78,E2 -3532.78} C_VEL
LIN {X 0,Y 544.572,Z 366.278,A -85,B 0,C 180,E1 -3533.612,E2 -3533.612} C_VEL
LIN {X 0,Y 544.579,Z 365.198,A -85,B 0,C 180,E1 -3534.392,E2 -3534.392} C_VEL
LIN {X 0,Y 544.641,Z 363.051,A -85,B 0,C 180,E1 -3535.41,E2 -3535.41} C_VEL
LIN {X 0,Y 544.694,Z 360.091,A -85,B 0,C 180,E1 -3536.432,E2 -3536.432} C_VEL
LIN {X 0,Y 544.697,Z 355.296,A -85,B 0,C 180,E1 -3537.677,E2 -3537.677} C_VEL
LIN {X 0,Y 544.762,Z 350.314,A -85,B 0,C 180,E1 -3538.687,E2 -3538.687} C_VEL
LIN {X 0,Y 544.887,Z 343.713,A -85,B 0,C 180,E1 -3539.774,E2 -3539.774} C_VEL
LIN {X 0,Y 545.031,Z 335.773,A -85,B 0,C 180,E1 -3540.835,E2 -3540.835} C_VEL
LIN {X 0,Y 545.25,Z 325.788,A -85,B 0,C 180,E1 -3541.902,E2 -3541.902} C_VEL
LIN {X 0,Y 545.415,Z 315.825,A -85,B 0,C 180,E1 -3542.765,E2 -3542.765} C_VEL
LIN {X 0,Y 545.664,Z 304.474,A -85,B 0,C 180,E1 -3543.55,E2 -3543.55} C_VEL
LIN {X 0,Y 545.872,Z 292.973,A -85,B 0,C 180,E1 -3544.171,E2 -3544.171} C_VEL
LIN {X 0,Y 546.029,Z 280.085,A -85,B 0,C 180,E1 -3544.696,E2 -3544.696} C_VEL
LIN {X 0,Y 546.138,Z 266.778,A -85,B 0,C 180,E1 -3545.061,E2 -3545.061} C_VEL
LIN {X 0,Y 546.255,Z 247.99,A -85,B 0,C 180,E1 -3545.349,E2 -3545.349} C_VEL
LIN {X 0,Y 546.455,Z 163.839,A -85,B 0,C 180,E1 -3546.462,E2 -3546.462} C_VEL
LIN {X 0,Y 545.232,Z 156.919,A -85,B 0,C 180,E1 -3546.598,E2 -3546.598} C_VEL
LIN {X 0,Y 545.417,Z 143.138,A -85,B 0,C 180,E1 -3549.153,E2 -3549.153} C_VEL
LIN {X 0,Y 545.373,Z 132.583,A -85,B 0,C 180,E1 -3551.088,E2 -3551.088} C_VEL
LIN {X 0,Y 545.133,Z 130.583,A -85,B 0,C 180,E1 -3551.477,E2 -3551.477} C_VEL
LIN {X 0,Y 545.055,Z 130.594,A -85,B 0,C 180,E1 -3554.13,E2 -3554.13} C_VEL
LIN {X 0,Y 545.083,Z 130.582,A -85,B 0,C 180,E1 -3556.895,E2 -3556.895} C_VEL
LIN {X 0,Y 545.09,Z 130.591,A -85,B 0,C 180,E1 -3559.861,E2 -3559.861} C_VEL
LIN {X 0,Y 545.068,Z 130.588,A -85,B 0,C 180,E1 -3563.075,E2 -3563.075} C_VEL
LIN {X 0,Y 545.064,Z 130.585,A -85,B 0,C 180,E1 -3566.329,E2 -3566.329} C_VEL
LIN {X 0,Y 545.064,Z 130.587,A -85,B 0,C 180,E1 -3568.953,E2 -3568.953} C_VEL
LIN {X 0,Y 545.1,Z 130.588,A -85,B 0,C 180,E1 -3571.508,E2 -3571.508} C_VEL
LIN {X 0,Y 545.094,Z 130.582,A -85,B 0,C 180,E1 -3574.492,E2 -3574.492} C_VEL
LIN {X 0,Y 545.038,Z 130.597,A -85,B 0,C 180,E1 -3577.243,E2 -3577.243} C_VEL
LIN {X 0,Y 545.116,Z 130.579,A -85,B 0,C 180,E1 -3580.416,E2 -3580.416} C_VEL
LIN {X 0,Y 545.056,Z 130.588,A -85,B 0,C 180,E1 -3583.521,E2 -3583.521} C_VEL
LIN {X 0,Y 545.085,Z 130.581,A -85,B 0,C 180,E1 -3585.82,E2 -3585.82} C_VEL
LIN {X 0,Y 545.119,Z 130.587,A -85,B 0,C 180,E1 -3588.85,E2 -3588.85} C_VEL
LIN {X 0,Y 545.098,Z 130.579,A -85,B 0,C 180,E1 -3591.847,E2 -3591.847} C_VEL
LIN {X 0,Y 545.199,Z 130.571,A -85,B 0,C 180,E1 -3594.824,E2 -3594.824} C_VEL
LIN {X 0,Y 545.196,Z 130.568,A -85,B 0,C 180,E1 -3597.784,E2 -3597.784} C_VEL
LIN {X 0,Y 545.209,Z 130.568,A -85,B 0,C 180,E1 -3600.739,E2 -3600.739} C_VEL
LIN {X 0,Y 545.155,Z 130.574,A -85,B 0,C 180,E1 -3602.956,E2 -3602.956} C_VEL
LIN {X 0,Y 545.137,Z 130.577,A -85,B 0,C 180,E1 -3605.92,E2 -3605.92} C_VEL
LIN {X 0,Y 545.097,Z 130.58,A -85,B 0,C 180,E1 -3608.901,E2 -3608.901} C_VEL
LIN {X 0,Y 545.103,Z 130.584,A -85,B 0,C 180,E1 -3611.905,E2 -3611.905} C_VEL
LIN {X 0,Y 545.082,Z 130.582,A -85,B 0,C 180,E1 -3614.944,E2 -3614.944} C_VEL
LIN {X 0,Y 545.049,Z 130.593,A -85,B 0,C 180,E1 -3618.027,E2 -3618.027} C_VEL
LIN {X 0,Y 545.035,Z 130.588,A -85,B 0,C 180,E1 -3620.375,E2 -3620.375} C_VEL
LIN {X 0,Y 544.991,Z 130.593,A -85,B 0,C 180,E1 -3622.76,E2 -3622.76} C_VEL
LIN {X 0,Y 545.037,Z 130.596,A -85,B 0,C 180,E1 -3625.495,E2 -3625.495} C_VEL
LIN {X 0,Y 545.034,Z 130.588,A -85,B 0,C 180,E1 -3628.497,E2 -3628.497} C_VEL
LIN {X 0,Y 545.045,Z 130.592,A -85,B 0,C 180,E1 -3631.676,E2 -3631.676} C_VEL
LIN {X 0,Y 545.039,Z 130.587,A -85,B 0,C 180,E1 -3634.567,E2 -3634.567} C_VEL
LIN {X 0,Y 545.003,Z 130.598,A -85,B 0,C 180,E1 -3637.307,E2 -3637.307} C_VEL
LIN {X 0,Y 545.009,Z 130.592,A -85,B 0,C 180,E1 -3640.148,E2 -3640.148} C_VEL
LIN {X 0,Y 545.018,Z 130.598,A -85,B 0,C 180,E1 -3643.113,E2 -3643.113} C_VEL
LIN {X 0,Y 545.027,Z 130.592,A -85,B 0,C 180,E1 -3646.229,E2 -3646.229} C_VEL
LIN {X 0,Y 545.013,Z 130.6,A -85,B 0,C 180,E1 -3648.879,E2 -3648.879} C_VEL
LIN {X 0,Y 545.045,Z 130.588,A -85,B 0,C 180,E1 -3651.762,E2 -3651.762} C_VEL
LIN {X 0,Y 545.025,Z 130.597,A -85,B 0,C 180,E1 -3654.531,E2 -3654.531} C_VEL
LIN {X 0,Y 545.063,Z 130.587,A -85,B 0,C 180,E1 -3657.211,E2 -3657.211} C_VEL
LIN {X 0,Y 545.064,Z 130.587,A -85,B 0,C 180,E1 -3659.81,E2 -3659.81} C_VEL
LIN {X 0,Y 545.037,Z 130.592,A -85,B 0,C 180,E1 -3662.839,E2 -3662.839} C_VEL
LIN {X 0,Y 545.068,Z 130.594,A -85,B 0,C 180,E1 -3665.998,E2 -3665.998} C_VEL
LIN {X 0,Y 546.156,Z 137.466,A -85,B 0,C 180,E1 -3667.092,E2 -3667.092} C_VEL
LIN {X 0,Y 545.864,Z 156.303,A -85,B 0,C 180,E1 -3669.907,E2 -3669.907} C_VEL
LIN {X 0,Y 545.536,Z 175.699,A -85,B 0,C 180,E1 -3672.764,E2 -3672.764} C_VEL
LIN {X 0,Y 545.328,Z 194.048,A -85,B 0,C 180,E1 -3675.44,E2 -3675.44} C_VEL
LIN {X 0,Y 546.476,Z 203.411,A -85,B 0,C 180,E1 -3675.596,E2 -3675.596} C_VEL
LIN {X 0,Y 546.179,Z 302.297,A -85,B 0,C 180,E1 -3676.916,E2 -3676.916} C_VEL
LIN {X 0,Y 546.056,Z 315.632,A -85,B 0,C 180,E1 -3677.244,E2 -3677.244} C_VEL
LIN {X 0,Y 545.857,Z 327.834,A -85,B 0,C 180,E1 -3677.688,E2 -3677.688} C_VEL
LIN {X 0,Y 545.684,Z 338.936,A -85,B 0,C 180,E1 -3678.228,E2 -3678.228} C_VEL
LIN {X 0,Y 545.504,Z 350.478,A -85,B 0,C 180,E1 -3678.951,E2 -3678.951} C_VEL
LIN {X 0,Y 545.248,Z 361.167,A -85,B 0,C 180,E1 -3679.792,E2 -3679.792} C_VEL
LIN {X 0,Y 545.088,Z 370.803,A -85,B 0,C 180,E1 -3680.725,E2 -3680.725} C_VEL
LIN {X 0,Y 544.947,Z 378.701,A -85,B 0,C 180,E1 -3681.658,E2 -3681.658} C_VEL
LIN {X 0,Y 544.824,Z 386.416,A -85,B 0,C 180,E1 -3682.775,E2 -3682.775} C_VEL
LIN {X 0,Y 544.777,Z 393.528,A -85,B 0,C 180,E1 -3684.076,E2 -3684.076} C_VEL
LIN {X 0,Y 544.629,Z 398.254,A -85,B 0,C 180,E1 -3685.189,E2 -3685.189} C_VEL
LIN {X 0,Y 544.669,Z 401.871,A -85,B 0,C 180,E1 -3686.301,E2 -3686.301} C_VEL
LIN {X 0,Y 544.65,Z 403.734,A -85,B 0,C 180,E1 -3687.042,E2 -3687.042} C_VEL
LIN {X 0,Y 544.546,Z 406.126,A -85,B 0,C 180,E1 -3688.521,E2 -3688.521} C_VEL
LIN {X 0,Y 544.542,Z 406.735,A -85,B 0,C 180,E1 -3689.261,E2 -3689.261} C_VEL
LIN {X 0,Y 544.541,Z 406.951,A -85,B 0,C 180,E1 -3690,E2 -3690} C_VEL
LIN {X 0,Y 544.542,Z 406.735,A -85,B 0,C 180,E1 -3690.74,E2 -3690.74} C_VEL
LIN {X 0,Y 544.572,Z 405.132,A -85,B 0,C 180,E1 -3692.219,E2 -3692.219} C_VEL
LIN {X 0,Y 544.651,Z 403.738,A -85,B 0,C 180,E1 -3692.959,E2 -3692.959} C_VEL
LIN {X 0,Y 544.684,Z 400.8,A -85,B 0,C 180,E1 -3694.07,E2 -3694.07} C_VEL
LIN {X 0,Y 544.654,Z 396.82,A -85,B 0,C 180,E1 -3695.183,E2 -3695.183} C_VEL
LIN {X 0,Y 544.73,Z 391.431,A -85,B 0,C 180,E1 -3696.348,E2 -3696.348} C_VEL
LIN {X 0,Y 544.86,Z 384.017,A -85,B 0,C 180,E1 -3697.598,E2 -3697.598} C_VEL
LIN {X 0,Y 545.001,Z 375.721,A -85,B 0,C 180,E1 -3698.715,E2 -3698.715} C_VEL
LIN {X 0,Y 545.148,Z 367.217,A -85,B 0,C 180,E1 -3699.648,E2 -3699.648} C_VEL
LIN {X 0,Y 545.368,Z 356.712,A -85,B 0,C 180,E1 -3700.582,E2 -3700.582} C_VEL
LIN {X 0,Y 545.578,Z 345.139,A -85,B 0,C 180,E1 -3701.407,E2 -3701.407} C_VEL
LIN {X 0,Y 545.773,Z 334.925,A -85,B 0,C 180,E1 -3701.985,E2 -3701.985} C_VEL
LIN {X 0,Y 545.949,Z 323.229,A -85,B 0,C 180,E1 -3702.5,E2 -3702.5} C_VEL
LIN {X 0,Y 546.117,Z 309.753,A -85,B 0,C 180,E1 -3702.921,E2 -3702.921} C_VEL
LIN {X 0,Y 546.277,Z 296.402,A -85,B 0,C 180,E1 -3703.177,E2 -3703.177} C_VEL
LIN {X 0,Y 546.341,Z 200.961,A -85,B 0,C 180,E1 -3704.441,E2 -3704.441} C_VEL
LIN {X 0,Y 545.324,Z 193.989,A -85,B 0,C 180,E1 -3704.58,E2 -3704.58} C_VEL
LIN {X 0,Y 545.572,Z 174.262,A -85,B 0,C 180,E1 -3707.468,E2 -3707.468} C_VEL
LIN {X 0,Y 545.974,Z 153.519,A -85,B 0,C 180,E1 -3710.535,E2 -3710.535} C_VEL
LIN {X 0,Y 546.206,Z 137.775,A -85,B 0,C 180,E1 -3712.907,E2 -3712.907} C_VEL
LIN {X 0,Y 545.059,Z 130.591,A -85,B 0,C 180,E1 -3714.074,E2 -3714.074} C_VEL
LIN {X 0,Y 545.04,Z 130.591,A -85,B 0,C 180,E1 -3717.161,E2 -3717.161} C_VEL
LIN {X 0,Y 545.066,Z 130.588,A -85,B 0,C 180,E1 -3720.19,E2 -3720.19} C_VEL
LIN {X 0,Y 545.074,Z 130.585,A -85,B 0,C 180,E1 -3723.061,E2 -3723.061} C_VEL
LIN {X 0,Y 545.025,Z 130.596,A -85,B 0,C 180,E1 -3725.671,E2 -3725.671} C_VEL
LIN {X 0,Y 545.05,Z 130.586,A -85,B 0,C 180,E1 -3728.238,E2 -3728.238} C_VEL
LIN {X 0,Y 545.032,Z 130.593,A -85,B 0,C 180,E1 -3731.12,E2 -3731.12} C_VEL
LIN {X 0,Y 545.036,Z 130.588,A -85,B 0,C 180,E1 -3734.132,E2 -3734.132} C_VEL
LIN {X 0,Y 545.022,Z 130.593,A -85,B 0,C 180,E1 -3736.887,E2 -3736.887} C_VEL
LIN {X 0,Y 545.067,Z 130.585,A -85,B 0,C 180,E1 -3739.857,E2 -3739.857} C_VEL
LIN {X 0,Y 545.069,Z 130.593,A -85,B 0,C 180,E1 -3743.075,E2 -3743.075} C_VEL
LIN {X 0,Y 545.051,Z 130.587,A -85,B 0,C 180,E1 -3746.327,E2 -3746.327} C_VEL
LIN {X 0,Y 545.04,Z 130.597,A -85,B 0,C 180,E1 -3748.95,E2 -3748.95} C_VEL
LIN {X 0,Y 545.044,Z 130.588,A -85,B 0,C 180,E1 -3751.504,E2 -3751.504} C_VEL
LIN {X 0,Y 545.049,Z 130.586,A -85,B 0,C 180,E1 -3753.997,E2 -3753.997} C_VEL
LIN {X 0,Y 545.058,Z 130.589,A -85,B 0,C 180,E1 -3756.439,E2 -3756.439} C_VEL
LIN {X 0,Y 545.04,Z 130.595,A -85,B 0,C 180,E1 -3758.835,E2 -3758.835} C_VEL
LIN {X 0,Y 545.047,Z 130.589,A -85,B 0,C 180,E1 -3761.194,E2 -3761.194} C_VEL
LIN {X 0,Y 545.037,Z 130.592,A -85,B 0,C 180,E1 -3764.288,E2 -3764.288} C_VEL
LIN {X 0,Y 545.047,Z 130.595,A -85,B 0,C 180,E1 -3766.579,E2 -3766.579} C_VEL
LIN {X 0,Y 545.121,Z 130.581,A -85,B 0,C 180,E1 -3768.849,E2 -3768.849} C_VEL
LIN {X 0,Y 545.089,Z 130.583,A -85,B 0,C 180,E1 -3771.846,E2 -3771.846} C_VEL
LIN {X 0,Y 545.167,Z 130.574,A -85,B 0,C 180,E1 -3774.822,E2 -3774.822} C_VEL
LIN {X 0,Y 545.193,Z 130.57,A -85,B 0,C 180,E1 -3777.783,E2 -3777.783} C_VEL
LIN {X 0,Y 545.195,Z 130.574,A -85,B 0,C 180,E1 -3779.999,E2 -3779.999} C_VEL
LIN {X 0,Y 545.148,Z 130.574,A -85,B 0,C 180,E1 -3782.955,E2 -3782.955} C_VEL
LIN {X 0,Y 545.127,Z 130.583,A -85,B 0,C 180,E1 -3785.919,E2 -3785.919} C_VEL
LIN {X 0,Y 545.071,Z 130.583,A -85,B 0,C 180,E1 -3788.9,E2 -3788.9} C_VEL
LIN {X 0,Y 545.069,Z 130.593,A -85,B 0,C 180,E1 -3791.905,E2 -3791.905} C_VEL
LIN {X 0,Y 545.078,Z 130.582,A -85,B 0,C 180,E1 -3794.943,E2 -3794.943} C_VEL
LIN {X 0,Y 545.044,Z 130.592,A -85,B 0,C 180,E1 -3798.026,E2 -3798.026} C_VEL
LIN {X 0,Y 545.031,Z 130.589,A -85,B 0,C 180,E1 -3800.374,E2 -3800.374} C_VEL
LIN {X 0,Y 544.992,Z 130.593,A -85,B 0,C 180,E1 -3802.759,E2 -3802.759} C_VEL
LIN {X 0,Y 545.036,Z 130.595,A -85,B 0,C 180,E1 -3805.494,E2 -3805.494} C_VEL
LIN {X 0,Y 545.032,Z 130.588,A -85,B 0,C 180,E1 -3808.495,E2 -3808.495} C_VEL
LIN {X 0,Y 545.043,Z 130.593,A -85,B 0,C 180,E1 -3811.675,E2 -3811.675} C_VEL
LIN {X 0,Y 545.044,Z 130.587,A -85,B 0,C 180,E1 -3814.565,E2 -3814.565} C_VEL
LIN {X 0,Y 545.056,Z 130.589,A -85,B 0,C 180,E1 -3816.969,E2 -3816.969} C_VEL
LIN {X 0,Y 544.346,Z 130.683,A -85,B 0,C 180,E1 -3817.585,E2 -3817.585} C_VEL
LIN {X 0,Y 541.48,Z 131.039,A -85,B 0,C 180,E1 -3818.586,E2 -3818.586} C_VEL
LIN {X 0,Y 539.084,Z 131.337,A -85,B 0,C 180,E1 -3819.392,E2 -3819.392} C_VEL
LIN {X 0,Y 538.06,Z 131.458,A -85,B 0,C 180,E1 -3820.014,E2 -3820.014} C_VEL
LIN {X 0,Y 537.977,Z 131.467,A -85,B 0,C 180,E1 -3820.224,E2 -3820.224} C_VEL
LIN {X 0,Y 537.966,Z 131.474,A -85,B 0,C 180,E1 -3822.98,E2 -3822.98} C_VEL
LIN {X 0,Y 537.997,Z 131.465,A -85,B 0,C 180,E1 -3825.928,E2 -3825.928} C_VEL
LIN {X 0,Y 537.996,Z 131.47,A -85,B 0,C 180,E1 -3829.258,E2 -3829.258} C_VEL
LIN {X 0,Y 537.981,Z 131.467,A -85,B 0,C 180,E1 -3832.121,E2 -3832.121} C_VEL
LIN {X 0,Y 537.98,Z 131.476,A -85,B 0,C 180,E1 -3834.914,E2 -3834.914} C_VEL
LIN {X 0,Y 538.005,Z 131.464,A -85,B 0,C 180,E1 -3837.616,E2 -3837.616} C_VEL
LIN {X 0,Y 537.973,Z 131.469,A -85,B 0,C 180,E1 -3840.236,E2 -3840.236} C_VEL
LIN {X 0,Y 538,Z 131.472,A -85,B 0,C 180,E1 -3842.792,E2 -3842.792} C_VEL
LIN {X 0,Y 537.974,Z 131.469,A -85,B 0,C 180,E1 -3845.289,E2 -3845.289} C_VEL
LIN {X 0,Y 537.988,Z 131.468,A -85,B 0,C 180,E1 -3848.047,E2 -3848.047} C_VEL
LIN {X 0,Y 537.998,Z 131.468,A -85,B 0,C 180,E1 -3850.938,E2 -3850.938} C_VEL
LIN {X 0,Y 537.955,Z 131.47,A -85,B 0,C 180,E1 -3853.297,E2 -3853.297} C_VEL
LIN {X 0,Y 538.033,Z 131.46,A -85,B 0,C 180,E1 -3855.63,E2 -3855.63} C_VEL
LIN {X 0,Y 538.015,Z 131.466,A -85,B 0,C 180,E1 -3858.7,E2 -3858.7} C_VEL
LIN {X 0,Y 538.026,Z 131.463,A -85,B 0,C 180,E1 -3861.738,E2 -3861.738} C_VEL
LIN {X 0,Y 538.114,Z 131.452,A -85,B 0,C 180,E1 -3864.754,E2 -3864.754} C_VEL
LIN {X 0,Y 538.155,Z 131.45,A -85,B 0,C 180,E1 -3867.755,E2 -3867.755} C_VEL
LIN {X 0,Y 538.151,Z 131.455,A -85,B 0,C 180,E1 -3870,E2 -3870} C_VEL
LIN {X 0,Y 538.125,Z 131.586,A -85,B 0,C 180,E1 -3872.479,E2 -3872.479} C_VEL
LIN {X 0,Y 538.392,Z 138.219,A -85,B 0,C 180,E1 -3873.742,E2 -3873.742} C_VEL
LIN {X 0,Y 538.25,Z 154.278,A -85,B 0,C 180,E1 -3876.749,E2 -3876.749} C_VEL
LIN {X 0,Y 538.202,Z 157.317,A -85,B 0,C 180,E1 -3877.31,E2 -3877.31} C_VEL
LIN {X 0,Y 539.636,Z 165.348,A -85,B 0,C 180,E1 -3877.46,E2 -3877.46} C_VEL
LIN {X 0,Y 539.28,Z 264.48,A -85,B 0,C 180,E1 -3878.808,E2 -3878.808} C_VEL
LIN {X 0,Y 539.09,Z 277.605,A -85,B 0,C 180,E1 -3879.142,E2 -3879.142} C_VEL
LIN {X 0,Y 538.972,Z 290.14,A -85,B 0,C 180,E1 -3879.617,E2 -3879.617} C_VEL
LIN {X 0,Y 538.761,Z 302.154,A -85,B 0,C 180,E1 -3880.238,E2 -3880.238} C_VEL
LIN {X 0,Y 538.506,Z 313.665,A -85,B 0,C 180,E1 -3881.003,E2 -3881.003} C_VEL
LIN {X 0,Y 538.314,Z 323.48,A -85,B 0,C 180,E1 -3881.817,E2 -3881.817} C_VEL
LIN {X 0,Y 538.079,Z 333.34,A -85,B 0,C 180,E1 -3882.829,E2 -3882.829} C_VEL
LIN {X 0,Y 537.913,Z 342.394,A -85,B 0,C 180,E1 -3883.987,E2 -3883.987} C_VEL
LIN {X 0,Y 537.747,Z 349.686,A -85,B 0,C 180,E1 -3885.152,E2 -3885.152} C_VEL
LIN {X 0,Y 537.654,Z 355.47,A -85,B 0,C 180,E1 -3886.322,E2 -3886.322} C_VEL
LIN {X 0,Y 537.583,Z 360.011,A -85,B 0,C 180,E1 -3887.499,E2 -3887.499} C_VEL
LIN {X 0,Y 537.545,Z 362.408,A -85,B 0,C 180,E1 -3888.287,E2 -3888.287} C_VEL
LIN {X 0,Y 537.487,Z 365.516,A -85,B 0,C 180,E1 -3889.707,E2 -3889.707} C_VEL
LIN {X 0,Y 537.488,Z 366.765,A -85,B 0,C 180,E1 -3890.673,E2 -3890.673} C_VEL
LIN {X 0,Y 537.472,Z 367.401,A -85,B 0,C 180,E1 -3891.816,E2 -3891.816} C_VEL
LIN {X 0,Y 537.466,Z 367.039,A -85,B 0,C 180,E1 -3893.097,E2 -3893.097} C_VEL
LIN {X 0,Y 537.482,Z 366.217,A -85,B 0,C 180,E1 -3893.913,E2 -3893.913} C_VEL
LIN {X 0,Y 537.495,Z 364.874,A -85,B 0,C 180,E1 -3894.735,E2 -3894.735} C_VEL
LIN {X 0,Y 537.567,Z 361.932,A -85,B 0,C 180,E1 -3895.974,E2 -3895.974} C_VEL
LIN {X 0,Y 537.629,Z 357.581,A -85,B 0,C 180,E1 -3897.265,E2 -3897.265} C_VEL
LIN {X 0,Y 537.692,Z 352.177,A -85,B 0,C 180,E1 -3898.472,E2 -3898.472} C_VEL
LIN {X 0,Y 537.814,Z 344.634,A -85,B 0,C 180,E1 -3899.774,E2 -3899.774} C_VEL
LIN {X 0,Y 537.981,Z 336.851,A -85,B 0,C 180,E1 -3900.847,E2 -3900.847} C_VEL
LIN {X 0,Y 538.229,Z 327.123,A -85,B 0,C 180,E1 -3901.926,E2 -3901.926} C_VEL
LIN {X 0,Y 538.399,Z 317.372,A -85,B 0,C 180,E1 -3902.801,E2 -3902.801} C_VEL
LIN {X 0,Y 538.647,Z 306.857,A -85,B 0,C 180,E1 -3903.565,E2 -3903.565} C_VEL
LIN {X 0,Y 538.887,Z 295.546,A -85,B 0,C 180,E1 -3904.218,E2 -3904.218} C_VEL
LIN {X 0,Y 539.125,Z 283.671,A -85,B 0,C 180,E1 -3904.737,E2 -3904.737} C_VEL
LIN {X 0,Y 539.238,Z 271.046,A -85,B 0,C 180,E1 -3905.134,E2 -3905.134} C_VEL
LIN {X 0,Y 539.369,Z 258.495,A -85,B 0,C 180,E1 -3905.382,E2 -3905.382} C_VEL
LIN {X 0,Y 539.576,Z 164.633,A -85,B 0,C 180,E1 -3906.643,E2 -3906.643} C_VEL
LIN {X 0,Y 538.243,Z 157.174,A -85,B 0,C 180,E1 -3906.795,E2 -3906.795} C_VEL
LIN {X 0,Y 538.44,Z 141.181,A -85,B 0,C 180,E1 -3909.76,E2 -3909.76} C_VEL
LIN {X 0,Y 538.459,Z 134.546,A -85,B 0,C 180,E1 -3910.985,E2 -3910.985} C_VEL
LIN {X 0,Y 538.082,Z 131.462,A -85,B 0,C 180,E1 -3911.58,E2 -3911.58} C_VEL
LIN {X 0,Y 538.029,Z 131.463,A -85,B 0,C 180,E1 -3914.86,E2 -3914.86} C_VEL
LIN {X 0,Y 538.035,Z 131.467,A -85,B 0,C 180,E1 -3918.121,E2 -3918.121} C_VEL
LIN {X 0,Y 538.056,Z 131.46,A -85,B 0,C 180,E1 -3920.412,E2 -3920.412} C_VEL
LIN {X 0,Y 538.022,Z 131.466,A -85,B 0,C 180,E1 -3923.068,E2 -3923.068} C_VEL
LIN {X 0,Y 538.017,Z 131.468,A -85,B 0,C 180,E1 -3925.828,E2 -3925.828} C_VEL
LIN {X 0,Y 538.007,Z 131.464,A -85,B 0,C 180,E1 -3928.499,E2 -3928.499} C_VEL
LIN {X 0,Y 538.059,Z 131.461,A -85,B 0,C 180,E1 -3931.101,E2 -3931.101} C_VEL
LIN {X 0,Y 538.041,Z 131.465,A -85,B 0,C 180,E1 -3933.634,E2 -3933.634} C_VEL
LIN {X 0,Y 538.006,Z 131.464,A -85,B 0,C 180,E1 -3936.123,E2 -3936.123} C_VEL
LIN {X 0,Y 538.037,Z 131.466,A -85,B 0,C 180,E1 -3939.349,E2 -3939.349} C_VEL
LIN {X 0,Y 538.036,Z 131.462,A -85,B 0,C 180,E1 -3942.468,E2 -3942.468} C_VEL
LIN {X 0,Y 538.057,Z 131.458,A -85,B 0,C 180,E1 -3945.631,E2 -3945.631} C_VEL
LIN {X 0,Y 538.078,Z 131.462,A -85,B 0,C 180,E1 -3948.702,E2 -3948.702} C_VEL
LIN {X 0,Y 538.062,Z 131.455,A -85,B 0,C 180,E1 -3951.74,E2 -3951.74} C_VEL
LIN {X 0,Y 538.157,Z 131.449,A -85,B 0,C 180,E1 -3954.756,E2 -3954.756} C_VEL
LIN {X 0,Y 538.167,Z 131.443,A -85,B 0,C 180,E1 -3957.755,E2 -3957.755} C_VEL
LIN {X 0,Y 538.18,Z 131.444,A -85,B 0,C 180,E1 -3960.749,E2 -3960.749} C_VEL
LIN {X 0,Y 538.122,Z 131.45,A -85,B 0,C 180,E1 -3962.995,E2 -3962.995} C_VEL
LIN {X 0,Y 538.09,Z 131.456,A -85,B 0,C 180,E1 -3965.998,E2 -3965.998} C_VEL
LIN {X 0,Y 538.05,Z 131.458,A -85,B 0,C 180,E1 -3969.019,E2 -3969.019} C_VEL
LIN {X 0,Y 538.061,Z 131.463,A -85,B 0,C 180,E1 -3972.064,E2 -3972.064} C_VEL
LIN {X 0,Y 538.04,Z 131.459,A -85,B 0,C 180,E1 -3975.144,E2 -3975.144} C_VEL
LIN {X 0,Y 538.004,Z 131.467,A -85,B 0,C 180,E1 -3978.272,E2 -3978.272} C_VEL
LIN {X 0,Y 537.991,Z 131.464,A -85,B 0,C 180,E1 -3980.654,E2 -3980.654} C_VEL
LIN {X 0,Y 537.978,Z 131.468,A -85,B 0,C 180,E1 -3983.074,E2 -3983.074} C_VEL
LIN {X 0,Y 537.996,Z 131.471,A -85,B 0,C 180,E1 -3985.661,E2 -3985.661} C_VEL
LIN {X 0,Y 537.973,Z 131.47,A -85,B 0,C 180,E1 -3988.054,E2 -3988.054} C_VEL
LIN {X 0,Y 537.989,Z 131.464,A -85,B 0,C 180,E1 -3990.629,E2 -3990.629} C_VEL
LIN {X 0,Y 538.001,Z 131.473,A -85,B 0,C 180,E1 -3993.275,E2 -3993.275} C_VEL
LIN {X 0,Y 537.953,Z 131.471,A -85,B 0,C 180,E1 -3996.008,E2 -3996.008} C_VEL
LIN {X 0,Y 537.979,Z 131.471,A -85,B 0,C 180,E1 -3998.834,E2 -3998.834} C_VEL
LIN {X 0,Y 537.977,Z 131.469,A -85,B 0,C 180,E1 -4001.872,E2 -4001.872} C_VEL
LIN {X 0,Y 537.995,Z 131.474,A -85,B 0,C 180,E1 -4004.864,E2 -4004.864} C_VEL
LIN {X 0,Y 537.972,Z 131.474,A -85,B 0,C 180,E1 -4007.209,E2 -4007.209} C_VEL
LIN {X 0,Y 538.008,Z 131.469,A -85,B 0,C 180,E1 -4010.419,E2 -4010.419} C_VEL
LIN {X 0,Y 538.019,Z 131.464,A -85,B 0,C 180,E1 -4013.067,E2 -4013.067} C_VEL
LIN {X 0,Y 537.999,Z 131.466,A -85,B 0,C 180,E1 -4015.825,E2 -4015.825} C_VEL
LIN {X 0,Y 538.01,Z 131.471,A -85,B 0,C 180,E1 -4018.499,E2 -4018.499} C_VEL
LIN {X 0,Y 538.004,Z 131.466,A -85,B 0,C 180,E1 -4021.097,E2 -4021.097} C_VEL
LIN {X 0,Y 537.992,Z 131.469,A -85,B 0,C 180,E1 -4023.631,E2 -4023.631} C_VEL
LIN {X 0,Y 538.044,Z 131.605,A -85,B 0,C 180,E1 -4025.873,E2 -4025.873} C_VEL
LIN {X 0,Y 539.197,Z 138.501,A -85,B 0,C 180,E1 -4026.982,E2 -4026.982} C_VEL
LIN {X 0,Y 538.913,Z 156.427,A -85,B 0,C 180,E1 -4029.697,E2 -4029.697} C_VEL
LIN {X 0,Y 538.54,Z 175.419,A -85,B 0,C 180,E1 -4032.533,E2 -4032.533} C_VEL
LIN {X 0,Y 538.252,Z 193.773,A -85,B 0,C 180,E1 -4035.245,E2 -4035.245} C_VEL
LIN {X 0,Y 539.592,Z 203.831,A -85,B 0,C 180,E1 -4035.418,E2 -4035.418} C_VEL
LIN {X 0,Y 539.282,Z 301.972,A -85,B 0,C 180,E1 -4036.745,E2 -4036.745} C_VEL
LIN {X 0,Y 539.134,Z 315.326,A -85,B 0,C 180,E1 -4037.077,E2 -4037.077} C_VEL
LIN {X 0,Y 538.905,Z 327.537,A -85,B 0,C 180,E1 -4037.526,E2 -4037.526} C_VEL
LIN {X 0,Y 538.688,Z 339.457,A -85,B 0,C 180,E1 -4038.118,E2 -4038.118} C_VEL
LIN {X 0,Y 538.46,Z 351.49,A -85,B 0,C 180,E1 -4038.9,E2 -4038.9} C_VEL
LIN {X 0,Y 538.197,Z 361.962,A -85,B 0,C 180,E1 -4039.751,E2 -4039.751} C_VEL
LIN {X 0,Y 538.048,Z 370.526,A -85,B 0,C 180,E1 -4040.603,E2 -4040.603} C_VEL
LIN {X 0,Y 537.899,Z 378.428,A -85,B 0,C 180,E1 -4041.548,E2 -4041.548} C_VEL
LIN {X 0,Y 537.755,Z 386.145,A -85,B 0,C 180,E1 -4042.679,E2 -4042.679} C_VEL
LIN {X 0,Y 537.666,Z 393.259,A -85,B 0,C 180,E1 -4043.998,E2 -4043.998} C_VEL
LIN {X 0,Y 537.54,Z 397.989,A -85,B 0,C 180,E1 -4045.125,E2 -4045.125} C_VEL
LIN {X 0,Y 537.591,Z 401.608,A -85,B 0,C 180,E1 -4046.252,E2 -4046.252} C_VEL
LIN {X 0,Y 537.551,Z 403.472,A -85,B 0,C 180,E1 -4047.002,E2 -4047.002} C_VEL
LIN {X 0,Y 537.451,Z 405.865,A -85,B 0,C 180,E1 -4048.502,E2 -4048.502} C_VEL
LIN {X 0,Y 537.446,Z 406.475,A -85,B 0,C 180,E1 -4049.251,E2 -4049.251} C_VEL
LIN {X 0,Y 537.447,Z 406.692,A -85,B 0,C 180,E1 -4050,E2 -4050} C_VEL
LIN {X 0,Y 537.452,Z 405.869,A -85,B 0,C 180,E1 -4051.499,E2 -4051.499} C_VEL
LIN {X 0,Y 537.49,Z 404.874,A -85,B 0,C 180,E1 -4052.248,E2 -4052.248} C_VEL
LIN {X 0,Y 537.551,Z 403.479,A -85,B 0,C 180,E1 -4052.998,E2 -4052.998} C_VEL
LIN {X 0,Y 537.603,Z 400.542,A -85,B 0,C 180,E1 -4054.123,E2 -4054.123} C_VEL
LIN {X 0,Y 537.588,Z 396.561,A -85,B 0,C 180,E1 -4055.251,E2 -4055.251} C_VEL
LIN {X 0,Y 537.654,Z 390.466,A -85,B 0,C 180,E1 -4056.563,E2 -4056.563} C_VEL
LIN {X 0,Y 537.785,Z 383.754,A -85,B 0,C 180,E1 -4057.698,E2 -4057.698} C_VEL
LIN {X 0,Y 537.934,Z 375.456,A -85,B 0,C 180,E1 -4058.831,E2 -4058.831} C_VEL
LIN {X 0,Y 538.102,Z 366.95,A -85,B 0,C 180,E1 -4059.776,E2 -4059.776} C_VEL
LIN {X 0,Y 538.355,Z 356.442,A -85,B 0,C 180,E1 -4060.721,E2 -4060.721} C_VEL
LIN {X 0,Y 538.583,Z 345.248,A -85,B 0,C 180,E1 -4061.532,E2 -4061.532} C_VEL
LIN {X 0,Y 538.814,Z 334.649,A -85,B 0,C 180,E1 -4062.142,E2 -4062.142} C_VEL
LIN {X 0,Y 538.986,Z 322.943,A -85,B 0,C 180,E1 -4062.664,E2 -4062.664} C_VEL
LIN {X 0,Y 539.187,Z 309.456,A -85,B 0,C 180,E1 -4063.09,E2 -4063.09} C_VEL
LIN {X 0,Y 539.361,Z 296.069,A -85,B 0,C 180,E1 -4063.349,E2 -4063.349} C_VEL
LIN {X 0,Y 539.507,Z 201.998,A -85,B 0,C 180,E1 -4064.61,E2 -4064.61} C_VEL
LIN {X 0,Y 538.299,Z 193.79,A -85,B 0,C 180,E1 -4064.767,E2 -4064.767} C_VEL
LIN {X 0,Y 538.564,Z 175.605,A -85,B 0,C 180,E1 -4067.466,E2 -4067.466} C_VEL
LIN {X 0,Y 539.004,Z 154.594,A -85,B 0,C 180,E1 -4070.613,E2 -4070.613} C_VEL
LIN {X 0,Y 539.264,Z 138.864,A -85,B 0,C 180,E1 -4073.016,E2 -4073.016} C_VEL
LIN {X 0,Y 538.013,Z 131.469,A -85,B 0,C 180,E1 -4074.241,E2 -4074.241} C_VEL
LIN {X 0,Y 538.012,Z 131.467,A -85,B 0,C 180,E1 -4077.207,E2 -4077.207} C_VEL
LIN {X 0,Y 538.003,Z 131.473,A -85,B 0,C 180,E1 -4079.762,E2 -4079.762} C_VEL
LIN {X 0,Y 538.018,Z 131.462,A -85,B 0,C 180,E1 -4082.383,E2 -4082.383} C_VEL
LIN {X 0,Y 537.991,Z 131.468,A -85,B 0,C 180,E1 -4085.085,E2 -4085.085} C_VEL
LIN {X 0,Y 537.991,Z 131.469,A -85,B 0,C 180,E1 -4087.878,E2 -4087.878} C_VEL
LIN {X 0,Y 538.007,Z 131.465,A -85,B 0,C 180,E1 -4090.78,E2 -4090.78} C_VEL
LIN {X 0,Y 538.006,Z 131.464,A -85,B 0,C 180,E1 -4094.071,E2 -4094.071} C_VEL
LIN {X 0,Y 537.976,Z 131.473,A -85,B 0,C 180,E1 -4097.019,E2 -4097.019} C_VEL
LIN {X 0,Y 538.01,Z 131.472,A -85,B 0,C 180,E1 -4099.258,E2 -4099.258} C_VEL
LIN {X 0,Y 537.991,Z 131.465,A -85,B 0,C 180,E1 -4102.122,E2 -4102.122} C_VEL
LIN {X 0,Y 537.992,Z 131.472,A -85,B 0,C 180,E1 -4104.915,E2 -4104.915} C_VEL
LIN {X 0,Y 538.015,Z 131.464,A -85,B 0,C 180,E1 -4107.617,E2 -4107.617} C_VEL
LIN {X 0,Y 537.985,Z 131.467,A -85,B 0,C 180,E1 -4110.236,E2 -4110.236} C_VEL
LIN {X 0,Y 538.014,Z 131.47,A -85,B 0,C 180,E1 -4112.793,E2 -4112.793} C_VEL
LIN {X 0,Y 537.984,Z 131.469,A -85,B 0,C 180,E1 -4115.289,E2 -4115.289} C_VEL
LIN {X 0,Y 538.001,Z 131.465,A -85,B 0,C 180,E1 -4118.047,E2 -4118.047} C_VEL
LIN {X 0,Y 538.011,Z 131.468,A -85,B 0,C 180,E1 -4120.939,E2 -4120.939} C_VEL
LIN {X 0,Y 537.969,Z 131.469,A -85,B 0,C 180,E1 -4123.297,E2 -4123.297} C_VEL
LIN {X 0,Y 538.04,Z 131.459,A -85,B 0,C 180,E1 -4125.629,E2 -4125.629} C_VEL
LIN {X 0,Y 538.082,Z 131.46,A -85,B 0,C 180,E1 -4128.701,E2 -4128.701} C_VEL
LIN {X 0,Y 538.053,Z 131.458,A -85,B 0,C 180,E1 -4131.739,E2 -4131.739} C_VEL
LIN {X 0,Y 538.126,Z 131.452,A -85,B 0,C 180,E1 -4134.754,E2 -4134.754} C_VEL
LIN {X 0,Y 538.165,Z 131.446,A -85,B 0,C 180,E1 -4137.754,E2 -4137.754} C_VEL
LIN {X 0,Y 538.163,Z 131.45,A -85,B 0,C 180,E1 -4139.999,E2 -4139.999} C_VEL
LIN {X 0,Y 538.115,Z 131.45,A -85,B 0,C 180,E1 -4142.994,E2 -4142.994} C_VEL
LIN {X 0,Y 538.083,Z 131.462,A -85,B 0,C 180,E1 -4145.997,E2 -4145.997} C_VEL
LIN {X 0,Y 538.029,Z 131.46,A -85,B 0,C 180,E1 -4149.018,E2 -4149.018} C_VEL
LIN {X 0,Y 538.04,Z 131.466,A -85,B 0,C 180,E1 -4152.063,E2 -4152.063} C_VEL
LIN {X 0,Y 538.038,Z 131.46,A -85,B 0,C 180,E1 -4155.143,E2 -4155.143} C_VEL
LIN {X 0,Y 537.997,Z 131.467,A -85,B 0,C 180,E1 -4158.271,E2 -4158.271} C_VEL
LIN {X 0,Y 537.988,Z 131.466,A -85,B 0,C 180,E1 -4160.653,E2 -4160.653} C_VEL
LIN {X 0,Y 537.98,Z 131.468,A -85,B 0,C 180,E1 -4163.073,E2 -4163.073} C_VEL
LIN {X 0,Y 537.994,Z 131.473,A -85,B 0,C 180,E1 -4165.66,E2 -4165.66} C_VEL
LIN {X 0,Y 537.971,Z 131.47,A -85,B 0,C 180,E1 -4168.053,E2 -4168.053} C_VEL
LIN {X 0,Y 537.991,Z 131.465,A -85,B 0,C 180,E1 -4170.628,E2 -4170.628} C_VEL
LIN {X 0,Y 538.019,Z 131.469,A -85,B 0,C 180,E1 -4173.278,E2 -4173.278} C_VEL
LIN {X 0,Y 537.967,Z 131.469,A -85,B 0,C 180,E1 -4176.006,E2 -4176.006} C_VEL
LIN {X 0,Y 538.004,Z 131.466,A -85,B 0,C 180,E1 -4178.83,E2 -4178.83} C_VEL
LIN {X 0,Y 537.977,Z 131.467,A -85,B 0,C 180,E1 -4180.224,E2 -4180.224} C_VEL
LIN {X 0,Y 537.311,Z 131.555,A -85,B 0,C 180,E1 -4180.85,E2 -4180.85} C_VEL
LIN {X 0,Y 534.458,Z 131.913,A -85,B 0,C 180,E1 -4181.864,E2 -4181.864} C_VEL
LIN {X 0,Y 532.045,Z 132.216,A -85,B 0,C 180,E1 -4182.681,E2 -4182.681} C_VEL
LIN {X 0,Y 531.007,Z 132.342,A -85,B 0,C 180,E1 -4183.312,E2 -4183.312} C_VEL
LIN {X 0,Y 530.922,Z 132.35,A -85,B 0,C 180,E1 -4183.526,E2 -4183.526} C_VEL
LIN {X 0,Y 530.961,Z 132.343,A -85,B 0,C 180,E1 -4185.623,E2 -4185.623} C_VEL
LIN {X 0,Y 530.931,Z 132.353,A -85,B 0,C 180,E1 -4188.982,E2 -4188.982} C_VEL
LIN {X 0,Y 530.946,Z 132.345,A -85,B 0,C 180,E1 -4191.528,E2 -4191.528} C_VEL
LIN {X 0,Y 530.929,Z 132.347,A -85,B 0,C 180,E1 -4194.378,E2 -4194.378} C_VEL
LIN {X 0,Y 530.959,Z 132.346,A -85,B 0,C 180,E1 -4197.132,E2 -4197.132} C_VEL
LIN {X 0,Y 530.929,Z 132.345,A -85,B 0,C 180,E1 -4199.8,E2 -4199.8} C_VEL
LIN {X 0,Y 530.955,Z 132.347,A -85,B 0,C 180,E1 -4202.478,E2 -4202.478} C_VEL
LIN {X 0,Y 530.941,Z 132.348,A -85,B 0,C 180,E1 -4204.939,E2 -4204.939} C_VEL
LIN {X 0,Y 530.944,Z 132.347,A -85,B 0,C 180,E1 -4208.245,E2 -4208.245} C_VEL
LIN {X 0,Y 530.955,Z 132.349,A -85,B 0,C 180,E1 -4210.675,E2 -4210.675} C_VEL
LIN {X 0,Y 530.919,Z 132.348,A -85,B 0,C 180,E1 -4213.069,E2 -4213.069} C_VEL
LIN {X 0,Y 530.993,Z 132.337,A -85,B 0,C 180,E1 -4215.435,E2 -4215.435} C_VEL
LIN {X 0,Y 530.977,Z 132.345,A -85,B 0,C 180,E1 -4218.548,E2 -4218.548} C_VEL
LIN {X 0,Y 530.974,Z 132.341,A -85,B 0,C 180,E1 -4221.628,E2 -4221.628} C_VEL
LIN {X 0,Y 531.075,Z 132.329,A -85,B 0,C 180,E1 -4224.685,E2 -4224.685} C_VEL
LIN {X 0,Y 531.126,Z 132.326,A -85,B 0,C 180,E1 -4227.725,E2 -4227.725} C_VEL
LIN {X 0,Y 531.12,Z 132.331,A -85,B 0,C 180,E1 -4230,E2 -4230} C_VEL
LIN {X 0,Y 531.1,Z 132.492,A -85,B 0,C 180,E1 -4232.37,E2 -4232.37} C_VEL
LIN {X 0,Y 531.403,Z 139.848,A -85,B 0,C 180,E1 -4233.791,E2 -4233.791} C_VEL
LIN {X 0,Y 531.237,Z 156.003,A -85,B 0,C 180,E1 -4236.838,E2 -4236.838} C_VEL
LIN {X 0,Y 531.216,Z 157.417,A -85,B 0,C 180,E1 -4237.102,E2 -4237.102} C_VEL
LIN {X 0,Y 532.816,Z 166.758,A -85,B 0,C 180,E1 -4237.285,E2 -4237.285} C_VEL
LIN {X 0,Y 532.391,Z 264.787,A -85,B 0,C 180,E1 -4238.636,E2 -4238.636} C_VEL
LIN {X 0,Y 532.174,Z 277.915,A -85,B 0,C 180,E1 -4238.975,E2 -4238.975} C_VEL
LIN {X 0,Y 532.039,Z 290.439,A -85,B 0,C 180,E1 -4239.456,E2 -4239.456} C_VEL
LIN {X 0,Y 531.812,Z 302.44,A -85,B 0,C 180,E1 -4240.084,E2 -4240.084} C_VEL
LIN {X 0,Y 531.545,Z 313.942,A -85,B 0,C 180,E1 -4240.86,E2 -4240.86} C_VEL
LIN {X 0,Y 531.333,Z 323.418,A -85,B 0,C 180,E1 -4241.654,E2 -4241.654} C_VEL
LIN {X 0,Y 531.082,Z 332.789,A -85,B 0,C 180,E1 -4242.612,E2 -4242.612} C_VEL
LIN {X 0,Y 530.863,Z 341.985,A -85,B 0,C 180,E1 -4243.786,E2 -4243.786} C_VEL
LIN {X 0,Y 530.71,Z 349.801,A -85,B 0,C 180,E1 -4245.035,E2 -4245.035} C_VEL
LIN {X 0,Y 530.592,Z 355.322,A -85,B 0,C 180,E1 -4246.15,E2 -4246.15} C_VEL
LIN {X 0,Y 530.497,Z 360.393,A -85,B 0,C 180,E1 -4247.477,E2 -4247.477} C_VEL
LIN {X 0,Y 530.456,Z 363.448,A -85,B 0,C 180,E1 -4248.54,E2 -4248.54} C_VEL
LIN {X 0,Y 530.399,Z 365.985,A -85,B 0,C 180,E1 -4249.82,E2 -4249.82} C_VEL
LIN {X 0,Y 530.378,Z 367.286,A -85,B 0,C 180,E1 -4250.964,E2 -4250.964} C_VEL
LIN {X 0,Y 530.373,Z 367.688,A -85,B 0,C 180,E1 -4251.943,E2 -4251.943} C_VEL
LIN {X 0,Y 530.402,Z 367.039,A -85,B 0,C 180,E1 -4253.423,E2 -4253.423} C_VEL
LIN {X 0,Y 530.392,Z 366.015,A -85,B 0,C 180,E1 -4254.253,E2 -4254.253} C_VEL
LIN {X 0,Y 530.431,Z 364.529,A -85,B 0,C 180,E1 -4255.087,E2 -4255.087} C_VEL
LIN {X 0,Y 530.53,Z 361.271,A -85,B 0,C 180,E1 -4256.345,E2 -4256.345} C_VEL
LIN {X 0,Y 530.568,Z 356.684,A -85,B 0,C 180,E1 -4257.621,E2 -4257.621} C_VEL
LIN {X 0,Y 530.643,Z 351.312,A -85,B 0,C 180,E1 -4258.773,E2 -4258.773} C_VEL
LIN {X 0,Y 530.799,Z 344.175,A -85,B 0,C 180,E1 -4259.988,E2 -4259.988} C_VEL
LIN {X 0,Y 530.993,Z 336.216,A -85,B 0,C 180,E1 -4261.077,E2 -4261.077} C_VEL
LIN {X 0,Y 531.255,Z 326.423,A -85,B 0,C 180,E1 -4262.152,E2 -4262.152} C_VEL
LIN {X 0,Y 531.468,Z 316.233,A -85,B 0,C 180,E1 -4263.057,E2 -4263.057} C_VEL
LIN {X 0,Y 531.755,Z 305.346,A -85,B 0,C 180,E1 -4263.831,E2 -4263.831} C_VEL
LIN {X 0,Y 532.051,Z 293.349,A -85,B 0,C 180,E1 -4264.496,E2 -4264.496} C_VEL
LIN {X 0,Y 532.209,Z 281.175,A -85,B 0,C 180,E1 -4265.007,E2 -4265.007} C_VEL
LIN {X 0,Y 532.377,Z 268.701,A -85,B 0,C 180,E1 -4265.372,E2 -4265.372} C_VEL
LIN {X 0,Y 532.461,Z 253.155,A -85,B 0,C 180,E1 -4265.635,E2 -4265.635} C_VEL
LIN {X 0,Y 532.736,Z 165.567,A -85,B 0,C 180,E1 -4266.825,E2 -4266.825} C_VEL
LIN {X 0,Y 531.245,Z 157.42,A -85,B 0,C 180,E1 -4266.995,E2 -4266.995} C_VEL
LIN {X 0,Y 531.491,Z 140.67,A -85,B 0,C 180,E1 -4270.114,E2 -4270.114} C_VEL
LIN {X 0,Y 531.264,Z 133.744,A -85,B 0,C 180,E1 -4271.41,E2 -4271.41} C_VEL
LIN {X 0,Y 531.025,Z 132.341,A -85,B 0,C 180,E1 -4271.686,E2 -4271.686} C_VEL
LIN {X 0,Y 530.985,Z 132.343,A -85,B 0,C 180,E1 -4274.547,E2 -4274.547} C_VEL
LIN {X 0,Y 530.986,Z 132.348,A -85,B 0,C 180,E1 -4277.834,E2 -4277.834} C_VEL
LIN {X 0,Y 531.003,Z 132.338,A -85,B 0,C 180,E1 -4280.559,E2 -4280.559} C_VEL
LIN {X 0,Y 530.952,Z 132.351,A -85,B 0,C 180,E1 -4283.442,E2 -4283.442} C_VEL
LIN {X 0,Y 530.996,Z 132.338,A -85,B 0,C 180,E1 -4286.495,E2 -4286.495} C_VEL
LIN {X 0,Y 530.972,Z 132.347,A -85,B 0,C 180,E1 -4289.356,E2 -4289.356} C_VEL
LIN {X 0,Y 531.012,Z 132.336,A -85,B 0,C 180,E1 -4292.468,E2 -4292.468} C_VEL
LIN {X 0,Y 531.005,Z 132.341,A -85,B 0,C 180,E1 -4294.943,E2 -4294.943} C_VEL
LIN {X 0,Y 530.971,Z 132.341,A -85,B 0,C 180,E1 -4298.247,E2 -4298.247} C_VEL
LIN {X 0,Y 530.983,Z 132.342,A -85,B 0,C 180,E1 -4300.678,E2 -4300.678} C_VEL
LIN {X 0,Y 530.965,Z 132.348,A -85,B 0,C 180,E1 -4303.071,E2 -4303.071} C_VEL
LIN {X 0,Y 531.015,Z 132.336,A -85,B 0,C 180,E1 -4305.436,E2 -4305.436} C_VEL
LIN {X 0,Y 531.036,Z 132.337,A -85,B 0,C 180,E1 -4308.55,E2 -4308.55} C_VEL
LIN {X 0,Y 531.037,Z 132.33,A -85,B 0,C 180,E1 -4311.63,E2 -4311.63} C_VEL
LIN {X 0,Y 531.117,Z 132.327,A -85,B 0,C 180,E1 -4314.686,E2 -4314.686} C_VEL
LIN {X 0,Y 531.139,Z 132.319,A -85,B 0,C 180,E1 -4317.726,E2 -4317.726} C_VEL
LIN {X 0,Y 531.15,Z 132.319,A -85,B 0,C 180,E1 -4320.759,E2 -4320.759} C_VEL
LIN {X 0,Y 531.063,Z 132.329,A -85,B 0,C 180,E1 -4323.035,E2 -4323.035} C_VEL
LIN {X 0,Y 531.047,Z 132.334,A -85,B 0,C 180,E1 -4326.078,E2 -4326.078} C_VEL
LIN {X 0,Y 531.012,Z 132.334,A -85,B 0,C 180,E1 -4329.139,E2 -4329.139} C_VEL
LIN {X 0,Y 531.052,Z 132.33,A -85,B 0,C 180,E1 -4331.671,E2 -4331.671} C_VEL
LIN {X 0,Y 531.032,Z 132.332,A -85,B 0,C 180,E1 -4334.955,E2 -4334.955} C_VEL
LIN {X 0,Y 530.966,Z 132.342,A -85,B 0,C 180,E1 -4338.523,E2 -4338.523} C_VEL
LIN {X 0,Y 530.943,Z 132.343,A -85,B 0,C 180,E1 -4340.941,E2 -4340.941} C_VEL
LIN {X 0,Y 530.955,Z 132.345,A -85,B 0,C 180,E1 -4344.031,E2 -4344.031} C_VEL
LIN {X 0,Y 530.948,Z 132.341,A -85,B 0,C 180,E1 -4346.747,E2 -4346.747} C_VEL
LIN {X 0,Y 530.917,Z 132.354,A -85,B 0,C 180,E1 -4349.327,E2 -4349.327} C_VEL
LIN {X 0,Y 530.952,Z 132.343,A -85,B 0,C 180,E1 -4352.098,E2 -4352.098} C_VEL
LIN {X 0,Y 530.952,Z 132.344,A -85,B 0,C 180,E1 -4354.848,E2 -4354.848} C_VEL
LIN {X 0,Y 530.906,Z 132.351,A -85,B 0,C 180,E1 -4357.513,E2 -4357.513} C_VEL
LIN {X 0,Y 530.909,Z 132.35,A -85,B 0,C 180,E1 -4360.44,E2 -4360.44} C_VEL
LIN {X 0,Y 530.927,Z 132.348,A -85,B 0,C 180,E1 -4363.499,E2 -4363.499} C_VEL
LIN {X 0,Y 530.967,Z 132.343,A -85,B 0,C 180,E1 -4365.624,E2 -4365.624} C_VEL
LIN {X 0,Y 530.932,Z 132.352,A -85,B 0,C 180,E1 -4368.983,E2 -4368.983} C_VEL
LIN {X 0,Y 530.95,Z 132.344,A -85,B 0,C 180,E1 -4371.529,E2 -4371.529} C_VEL
LIN {X 0,Y 530.937,Z 132.349,A -85,B 0,C 180,E1 -4374.379,E2 -4374.379} C_VEL
LIN {X 0,Y 530.968,Z 132.343,A -85,B 0,C 180,E1 -4377.133,E2 -4377.133} C_VEL
LIN {X 0,Y 530.952,Z 132.345,A -85,B 0,C 180,E1 -4379.802,E2 -4379.802} C_VEL
LIN {X 0,Y 530.965,Z 132.349,A -85,B 0,C 180,E1 -4382.478,E2 -4382.478} C_VEL
LIN {X 0,Y 530.953,Z 132.349,A -85,B 0,C 180,E1 -4385.566,E2 -4385.566} C_VEL
LIN {X 0,Y 530.983,Z 132.538,A -85,B 0,C 180,E1 -4385.724,E2 -4385.724} C_VEL
LIN {X 0,Y 532.239,Z 139.537,A -85,B 0,C 180,E1 -4386.869,E2 -4386.869} C_VEL
LIN {X 0,Y 531.97,Z 156.786,A -85,B 0,C 180,E1 -4389.519,E2 -4389.519} C_VEL
LIN {X 0,Y 531.533,Z 176.456,A -85,B 0,C 180,E1 -4392.494,E2 -4392.494} C_VEL
LIN {X 0,Y 531.208,Z 193.435,A -85,B 0,C 180,E1 -4395.035,E2 -4395.035} C_VEL
LIN {X 0,Y 532.733,Z 204.966,A -85,B 0,C 180,E1 -4395.245,E2 -4395.245} C_VEL
LIN {X 0,Y 532.386,Z 301.645,A -85,B 0,C 180,E1 -4396.57,E2 -4396.57} C_VEL
LIN {X 0,Y 532.203,Z 315.019,A -85,B 0,C 180,E1 -4396.906,E2 -4396.906} C_VEL
LIN {X 0,Y 531.962,Z 327.24,A -85,B 0,C 180,E1 -4397.361,E2 -4397.361} C_VEL
LIN {X 0,Y 531.72,Z 339.602,A -85,B 0,C 180,E1 -4397.987,E2 -4397.987} C_VEL
LIN {X 0,Y 531.465,Z 351.207,A -85,B 0,C 180,E1 -4398.752,E2 -4398.752} C_VEL
LIN {X 0,Y 531.209,Z 361.683,A -85,B 0,C 180,E1 -4399.615,E2 -4399.615} C_VEL
LIN {X 0,Y 530.986,Z 370.249,A -85,B 0,C 180,E1 -4400.477,E2 -4400.477} C_VEL
LIN {X 0,Y 530.848,Z 378.155,A -85,B 0,C 180,E1 -4401.435,E2 -4401.435} C_VEL
LIN {X 0,Y 530.667,Z 385.875,A -85,B 0,C 180,E1 -4402.581,E2 -4402.581} C_VEL
LIN {X 0,Y 530.561,Z 392.991,A -85,B 0,C 180,E1 -4403.917,E2 -4403.917} C_VEL
LIN {X 0,Y 530.459,Z 397.724,A -85,B 0,C 180,E1 -4405.06,E2 -4405.06} C_VEL
LIN {X 0,Y 530.516,Z 401.345,A -85,B 0,C 180,E1 -4406.202,E2 -4406.202} C_VEL
LIN {X 0,Y 530.457,Z 403.21,A -85,B 0,C 180,E1 -4406.962,E2 -4406.962} C_VEL
LIN {X 0,Y 530.412,Z 404.608,A -85,B 0,C 180,E1 -4407.722,E2 -4407.722} C_VEL
LIN {X 0,Y 530.351,Z 406.215,A -85,B 0,C 180,E1 -4409.241,E2 -4409.241} C_VEL
LIN {X 0,Y 530.352,Z 406.433,A -85,B 0,C 180,E1 -4410,E2 -4410} C_VEL
LIN {X 0,Y 530.361,Z 405.61,A -85,B 0,C 180,E1 -4411.519,E2 -4411.519} C_VEL
LIN {X 0,Y 530.412,Z 404.616,A -85,B 0,C 180,E1 -4412.278,E2 -4412.278} C_VEL
LIN {X 0,Y 530.457,Z 403.221,A -85,B 0,C 180,E1 -4413.038,E2 -4413.038} C_VEL
LIN {X 0,Y 530.521,Z 400.283,A -85,B 0,C 180,E1 -4414.178,E2 -4414.178} C_VEL
LIN {X 0,Y 530.522,Z 396.302,A -85,B 0,C 180,E1 -4415.321,E2 -4415.321} C_VEL
LIN {X 0,Y 530.556,Z 390.792,A -85,B 0,C 180,E1 -4416.541,E2 -4416.541} C_VEL
LIN {X 0,Y 530.705,Z 383.491,A -85,B 0,C 180,E1 -4417.802,E2 -4417.802} C_VEL
LIN {X 0,Y 530.887,Z 375.192,A -85,B 0,C 180,E1 -4418.949,E2 -4418.949} C_VEL
LIN {X 0,Y 531.062,Z 366.684,A -85,B 0,C 180,E1 -4419.907,E2 -4419.907} C_VEL
LIN {X 0,Y 531.343,Z 356.173,A -85,B 0,C 180,E1 -4420.864,E2 -4420.864} C_VEL
LIN {X 0,Y 531.61,Z 344.372,A -85,B 0,C 180,E1 -4421.726,E2 -4421.726} C_VEL
LIN {X 0,Y 531.869,Z 332.437,A -85,B 0,C 180,E1 -4422.4,E2 -4422.4} C_VEL
LIN {X 0,Y 532.112,Z 320.052,A -85,B 0,C 180,E1 -4422.927,E2 -4422.927} C_VEL
LIN {X 0,Y 532.303,Z 307.325,A -85,B 0,C 180,E1 -4423.311,E2 -4423.311} C_VEL
LIN {X 0,Y 532.473,Z 292.172,A -85,B 0,C 180,E1 -4423.574,E2 -4423.574} C_VEL
LIN {X 0,Y 532.629,Z 202.676,A -85,B 0,C 180,E1 -4424.79,E2 -4424.79} C_VEL
LIN {X 0,Y 531.273,Z 193.513,A -85,B 0,C 180,E1 -4424.97,E2 -4424.97} C_VEL
LIN {X 0,Y 531.606,Z 174.386,A -85,B 0,C 180,E1 -4427.849,E2 -4427.849} C_VEL
LIN {X 0,Y 532.035,Z 154.363,A -85,B 0,C 180,E1 -4430.896,E2 -4430.896} C_VEL
LIN {X 0,Y 532.32,Z 139.947,A -85,B 0,C 180,E1 -4433.128,E2 -4433.128} C_VEL
LIN {X 0,Y 530.98,Z 132.345,A -85,B 0,C 180,E1 -4434.407,E2 -4434.407} C_VEL
LIN {X 0,Y 530.967,Z 132.348,A -85,B 0,C 180,E1 -4437.522,E2 -4437.522} C_VEL
LIN {X 0,Y 530.965,Z 132.343,A -85,B 0,C 180,E1 -4440.643,E2 -4440.643} C_VEL
LIN {X 0,Y 530.965,Z 132.348,A -85,B 0,C 180,E1 -4443.499,E2 -4443.499} C_VEL
LIN {X 0,Y 530.954,Z 132.342,A -85,B 0,C 180,E1 -4446.559,E2 -4446.559} C_VEL
LIN {X 0,Y 530.973,Z 132.349,A -85,B 0,C 180,E1 -4449.445,E2 -4449.445} C_VEL
LIN {X 0,Y 530.922,Z 132.346,A -85,B 0,C 180,E1 -4452.463,E2 -4452.463} C_VEL
LIN {X 0,Y 530.968,Z 132.347,A -85,B 0,C 180,E1 -4455.45,E2 -4455.45} C_VEL
LIN {X 0,Y 530.963,Z 132.342,A -85,B 0,C 180,E1 -4458.561,E2 -4458.561} C_VEL
LIN {X 0,Y 530.956,Z 132.345,A -85,B 0,C 180,E1 -4461.529,E2 -4461.529} C_VEL
LIN {X 0,Y 530.952,Z 132.343,A -85,B 0,C 180,E1 -4464.379,E2 -4464.379} C_VEL
LIN {X 0,Y 530.97,Z 132.347,A -85,B 0,C 180,E1 -4467.133,E2 -4467.133} C_VEL
LIN {X 0,Y 530.94,Z 132.344,A -85,B 0,C 180,E1 -4469.801,E2 -4469.801} C_VEL
LIN {X 0,Y 530.968,Z 132.343,A -85,B 0,C 180,E1 -4472.478,E2 -4472.478} C_VEL
LIN {X 0,Y 530.952,Z 132.35,A -85,B 0,C 180,E1 -4474.939,E2 -4474.939} C_VEL
LIN {X 0,Y 530.957,Z 132.344,A -85,B 0,C 180,E1 -4478.246,E2 -4478.246} C_VEL
LIN {X 0,Y 530.968,Z 132.349,A -85,B 0,C 180,E1 -4480.676,E2 -4480.676} C_VEL
LIN {X 0,Y 530.933,Z 132.348,A -85,B 0,C 180,E1 -4483.069,E2 -4483.069} C_VEL
LIN {X 0,Y 531.002,Z 132.336,A -85,B 0,C 180,E1 -4485.435,E2 -4485.435} C_VEL
LIN {X 0,Y 531.04,Z 132.34,A -85,B 0,C 180,E1 -4488.549,E2 -4488.549} C_VEL
LIN {X 0,Y 530.999,Z 132.337,A -85,B 0,C 180,E1 -4491.628,E2 -4491.628} C_VEL
LIN {X 0,Y 531.088,Z 132.329,A -85,B 0,C 180,E1 -4494.684,E2 -4494.684} C_VEL
LIN {X 0,Y 531.137,Z 132.321,A -85,B 0,C 180,E1 -4497.724,E2 -4497.724} C_VEL
LIN {X 0,Y 531.132,Z 132.325,A -85,B 0,C 180,E1 -4499.999,E2 -4499.999} C_VEL
LIN {X 0,Y 531.137,Z 132.327,A -85,B 0,C 180,E1 -4502.274,E2 -4502.274} C_VEL
LIN {X 0,Y 531.086,Z 132.326,A -85,B 0,C 180,E1 -4505.314,E2 -4505.314} C_VEL
LIN {X 0,Y 530.986,Z 132.342,A -85,B 0,C 180,E1 -4508.371,E2 -4508.371} C_VEL
LIN {X 0,Y 531.014,Z 132.339,A -85,B 0,C 180,E1 -4511.649,E2 -4511.649} C_VEL
LIN {X 0,Y 531.021,Z 132.334,A -85,B 0,C 180,E1 -4514.949,E2 -4514.949} C_VEL
LIN {X 0,Y 530.956,Z 132.342,A -85,B 0,C 180,E1 -4518.522,E2 -4518.522} C_VEL
LIN {X 0,Y 530.941,Z 132.344,A -85,B 0,C 180,E1 -4520.94,E2 -4520.94} C_VEL
LIN {X 0,Y 530.953,Z 132.346,A -85,B 0,C 180,E1 -4524.03,E2 -4524.03} C_VEL
LIN {X 0,Y 530.946,Z 132.343,A -85,B 0,C 180,E1 -4526.746,E2 -4526.746} C_VEL
LIN {X 0,Y 530.952,Z 132.348,A -85,B 0,C 180,E1 -4529.324,E2 -4529.324} C_VEL
LIN {X 0,Y 530.956,Z 132.343,A -85,B 0,C 180,E1 -4532.098,E2 -4532.098} C_VEL
LIN {X 0,Y 530.955,Z 132.344,A -85,B 0,C 180,E1 -4534.848,E2 -4534.848} C_VEL
LIN {X 0,Y 530.96,Z 132.347,A -85,B 0,C 180,E1 -4537.507,E2 -4537.507} C_VEL
LIN {X 0,Y 530.938,Z 132.344,A -85,B 0,C 180,E1 -4540.436,E2 -4540.436} C_VEL
LIN {X 0,Y 530.922,Z 132.35,A -85,B 0,C 180,E1 -4543.526,E2 -4543.526} C_VEL
LIN {X 0,Y 530.257,Z 132.43,A -85,B 0,C 180,E1 -4544.159,E2 -4544.159} C_VEL
LIN {X 0,Y 527.418,Z 132.791,A -85,B 0,C 180,E1 -4545.188,E2 -4545.188} C_VEL
LIN {X 0,Y 525.011,Z 133.092,A -85,B 0,C 180,E1 -4546.017,E2 -4546.017} C_VEL
LIN {X 0,Y 523.966,Z 133.219,A -85,B 0,C 180,E1 -4546.656,E2 -4546.656} C_VEL
LIN {X 0,Y 523.874,Z 133.228,A -85,B 0,C 180,E1 -4546.873,E2 -4546.873} C_VEL
LIN {X 0,Y 523.908,Z 133.22,A -85,B 0,C 180,E1 -4549.916,E2 -4549.916} C_VEL
LIN {X 0,Y 523.897,Z 133.229,A -85,B 0,C 180,E1 -4552.866,E2 -4552.866} C_VEL
LIN {X 0,Y 523.906,Z 133.22,A -85,B 0,C 180,E1 -4555.707,E2 -4555.707} C_VEL
LIN {X 0,Y 523.903,Z 133.224,A -85,B 0,C 180,E1 -4558.454,E2 -4558.454} C_VEL
LIN {X 0,Y 523.893,Z 133.225,A -85,B 0,C 180,E1 -4561.122,E2 -4561.122} C_VEL
LIN {X 0,Y 523.904,Z 133.221,A -85,B 0,C 180,E1 -4563.996,E2 -4563.996} C_VEL
LIN {X 0,Y 523.89,Z 133.226,A -85,B 0,C 180,E1 -4566.268,E2 -4566.268} C_VEL
LIN {X 0,Y 523.915,Z 133.225,A -85,B 0,C 180,E1 -4568.765,E2 -4568.765} C_VEL
LIN {X 0,Y 523.917,Z 133.219,A -85,B 0,C 180,E1 -4571.219,E2 -4571.219} C_VEL
LIN {X 0,Y 523.903,Z 133.23,A -85,B 0,C 180,E1 -4574.437,E2 -4574.437} C_VEL
LIN {X 0,Y 523.937,Z 133.217,A -85,B 0,C 180,E1 -4577.606,E2 -4577.606} C_VEL
LIN {X 0,Y 523.936,Z 133.219,A -85,B 0,C 180,E1 -4580.737,E2 -4580.737} C_VEL
LIN {X 0,Y 523.993,Z 133.213,A -85,B 0,C 180,E1 -4583.84,E2 -4583.84} C_VEL
LIN {X 0,Y 524.096,Z 133.201,A -85,B 0,C 180,E1 -4587.694,E2 -4587.694} C_VEL
LIN {X 0,Y 524.088,Z 133.206,A -85,B 0,C 180,E1 -4590,E2 -4590} C_VEL
LIN {X 0,Y 524.097,Z 133.291,A -85,B 0,C 180,E1 -4592.233,E2 -4592.233} C_VEL
LIN {X 0,Y 524.443,Z 140.566,A -85,B 0,C 180,E1 -4593.649,E2 -4593.649} C_VEL
LIN {X 0,Y 524.239,Z 157.541,A -85,B 0,C 180,E1 -4596.881,E2 -4596.881} C_VEL
LIN {X 0,Y 525.982,Z 167.942,A -85,B 0,C 180,E1 -4597.102,E2 -4597.102} C_VEL
LIN {X 0,Y 525.513,Z 265.083,A -85,B 0,C 180,E1 -4598.459,E2 -4598.459} C_VEL
LIN {X 0,Y 525.261,Z 278.228,A -85,B 0,C 180,E1 -4598.803,E2 -4598.803} C_VEL
LIN {X 0,Y 525.13,Z 290.718,A -85,B 0,C 180,E1 -4599.29,E2 -4599.29} C_VEL
LIN {X 0,Y 524.867,Z 302.726,A -85,B 0,C 180,E1 -4599.927,E2 -4599.927} C_VEL
LIN {X 0,Y 524.596,Z 314.214,A -85,B 0,C 180,E1 -4600.713,E2 -4600.713} C_VEL
LIN {X 0,Y 524.347,Z 324.569,A -85,B 0,C 180,E1 -4601.598,E2 -4601.598} C_VEL
LIN {X 0,Y 524.039,Z 333.895,A -85,B 0,C 180,E1 -4602.588,E2 -4602.588} C_VEL
LIN {X 0,Y 523.814,Z 342.95,A -85,B 0,C 180,E1 -4603.777,E2 -4603.777} C_VEL
LIN {X 0,Y 523.658,Z 349.931,A -85,B 0,C 180,E1 -4604.918,E2 -4604.918} C_VEL
LIN {X 0,Y 523.532,Z 355.146,A -85,B 0,C 180,E1 -4605.974,E2 -4605.974} C_VEL
LIN {X 0,Y 523.424,Z 359.894,A -85,B 0,C 180,E1 -4607.181,E2 -4607.181} C_VEL
LIN {X 0,Y 523.374,Z 363.478,A -85,B 0,C 180,E1 -4608.395,E2 -4608.395} C_VEL
LIN {X 0,Y 523.303,Z 366.451,A -85,B 0,C 180,E1 -4609.934,E2 -4609.934} C_VEL
LIN {X 0,Y 523.286,Z 367.738,A -85,B 0,C 180,E1 -4611.261,E2 -4611.261} C_VEL
LIN {X 0,Y 523.291,Z 367.959,A -85,B 0,C 180,E1 -4612.089,E2 -4612.089} C_VEL
LIN {X 0,Y 523.289,Z 367.683,A -85,B 0,C 180,E1 -4612.922,E2 -4612.922} C_VEL
LIN {X 0,Y 523.309,Z 366.617,A -85,B 0,C 180,E1 -4614.046,E2 -4614.046} C_VEL
LIN {X 0,Y 523.374,Z 364.057,A -85,B 0,C 180,E1 -4615.449,E2 -4615.449} C_VEL
LIN {X 0,Y 523.443,Z 360.491,A -85,B 0,C 180,E1 -4616.73,E2 -4616.73} C_VEL
LIN {X 0,Y 523.535,Z 355.582,A -85,B 0,C 180,E1 -4618.024,E2 -4618.024} C_VEL
LIN {X 0,Y 523.649,Z 349.429,A -85,B 0,C 180,E1 -4619.266,E2 -4619.266} C_VEL
LIN {X 0,Y 523.807,Z 342.171,A -85,B 0,C 180,E1 -4620.431,E2 -4620.431} C_VEL
LIN {X 0,Y 524.051,Z 333.664,A -85,B 0,C 180,E1 -4621.535,E2 -4621.535} C_VEL
LIN {X 0,Y 524.285,Z 324.131,A -85,B 0,C 180,E1 -4622.539,E2 -4622.539} C_VEL
LIN {X 0,Y 524.563,Z 313.843,A -85,B 0,C 180,E1 -4623.411,E2 -4623.411} C_VEL
LIN {X 0,Y 524.887,Z 301.872,A -85,B 0,C 180,E1 -4624.219,E2 -4624.219} C_VEL
LIN {X 0,Y 525.186,Z 289.913,A -85,B 0,C 180,E1 -4624.837,E2 -4624.837} C_VEL
LIN {X 0,Y 525.365,Z 276.82,A -85,B 0,C 180,E1 -4625.333,E2 -4625.333} C_VEL
LIN {X 0,Y 525.505,Z 264.063,A -85,B 0,C 180,E1 -4625.654,E2 -4625.654} C_VEL
LIN {X 0,Y 525.879,Z 166.294,A -85,B 0,C 180,E1 -4627.016,E2 -4627.016} C_VEL
LIN {X 0,Y 524.276,Z 157.662,A -85,B 0,C 180,E1 -4627.194,E2 -4627.194} C_VEL
LIN {X 0,Y 524.499,Z 141.609,A -85,B 0,C 180,E1 -4630.204,E2 -4630.204} C_VEL
LIN {X 0,Y 524.338,Z 135.501,A -85,B 0,C 180,E1 -4631.359,E2 -4631.359} C_VEL
LIN {X 0,Y 523.962,Z 133.221,A -85,B 0,C 180,E1 -4631.815,E2 -4631.815} C_VEL
LIN {X 0,Y 523.952,Z 133.218,A -85,B 0,C 180,E1 -4634.692,E2 -4634.692} C_VEL
LIN {X 0,Y 523.955,Z 133.223,A -85,B 0,C 180,E1 -4637.882,E2 -4637.882} C_VEL
LIN {X 0,Y 523.929,Z 133.219,A -85,B 0,C 180,E1 -4640.917,E2 -4640.917} C_VEL
LIN {X 0,Y 523.898,Z 133.229,A -85,B 0,C 180,E1 -4643.826,E2 -4643.826} C_VEL
LIN {X 0,Y 523.939,Z 133.217,A -85,B 0,C 180,E1 -4646.636,E2 -4646.636} C_VEL
LIN {X 0,Y 523.954,Z 133.222,A -85,B 0,C 180,E1 -4649.356,E2 -4649.356} C_VEL
LIN {X 0,Y 523.976,Z 133.212,A -85,B 0,C 180,E1 -4652.282,E2 -4652.282} C_VEL
LIN {X 0,Y 523.952,Z 133.217,A -85,B 0,C 180,E1 -4654.582,E2 -4654.582} C_VEL
LIN {X 0,Y 523.911,Z 133.227,A -85,B 0,C 180,E1 -4657.107,E2 -4657.107} C_VEL
LIN {X 0,Y 523.979,Z 133.212,A -85,B 0,C 180,E1 -4659.867,E2 -4659.867} C_VEL
LIN {X 0,Y 523.943,Z 133.222,A -85,B 0,C 180,E1 -4662.837,E2 -4662.837} C_VEL
LIN {X 0,Y 523.974,Z 133.216,A -85,B 0,C 180,E1 -4665.236,E2 -4665.236} C_VEL
LIN {X 0,Y 524.014,Z 133.209,A -85,B 0,C 180,E1 -4668.395,E2 -4668.395} C_VEL
LIN {X 0,Y 523.989,Z 133.208,A -85,B 0,C 180,E1 -4671.516,E2 -4671.516} C_VEL
LIN {X 0,Y 524.078,Z 133.205,A -85,B 0,C 180,E1 -4674.614,E2 -4674.614} C_VEL
LIN {X 0,Y 524.111,Z 133.194,A -85,B 0,C 180,E1 -4677.695,E2 -4677.695} C_VEL
LIN {X 0,Y 524.121,Z 133.194,A -85,B 0,C 180,E1 -4680.769,E2 -4680.769} C_VEL
LIN {X 0,Y 524.006,Z 133.207,A -85,B 0,C 180,E1 -4683.076,E2 -4683.076} C_VEL
LIN {X 0,Y 524.067,Z 133.197,A -85,B 0,C 180,E1 -4685.387,E2 -4685.387} C_VEL
LIN {X 0,Y 523.963,Z 133.216,A -85,B 0,C 180,E1 -4688.485,E2 -4688.485} C_VEL
LIN {X 0,Y 524.002,Z 133.208,A -85,B 0,C 180,E1 -4691.737,E2 -4691.737} C_VEL
LIN {X 0,Y 523.995,Z 133.209,A -85,B 0,C 180,E1 -4695.052,E2 -4695.052} C_VEL
LIN {X 0,Y 523.916,Z 133.226,A -85,B 0,C 180,E1 -4697.971,E2 -4697.971} C_VEL
LIN {X 0,Y 523.935,Z 133.216,A -85,B 0,C 180,E1 -4700.412,E2 -4700.412} C_VEL
LIN {X 0,Y 523.887,Z 133.222,A -85,B 0,C 180,E1 -4702.895,E2 -4702.895} C_VEL
LIN {X 0,Y 523.901,Z 133.227,A -85,B 0,C 180,E1 -4705.422,E2 -4705.422} C_VEL
LIN {X 0,Y 523.898,Z 133.224,A -85,B 0,C 180,E1 -4708.004,E2 -4708.004} C_VEL
LIN {X 0,Y 523.899,Z 133.221,A -85,B 0,C 180,E1 -4710.846,E2 -4710.846} C_VEL
LIN {X 0,Y 523.913,Z 133.221,A -85,B 0,C 180,E1 -4713.726,E2 -4713.726} C_VEL
LIN {X 0,Y 523.858,Z 133.227,A -85,B 0,C 180,E1 -4716.394,E2 -4716.394} C_VEL
LIN {X 0,Y 523.89,Z 133.23,A -85,B 0,C 180,E1 -4719.088,E2 -4719.088} C_VEL
LIN {X 0,Y 523.891,Z 133.224,A -85,B 0,C 180,E1 -4722.126,E2 -4722.126} C_VEL
LIN {X 0,Y 523.936,Z 133.222,A -85,B 0,C 180,E1 -4725.312,E2 -4725.312} C_VEL
LIN {X 0,Y 523.913,Z 133.229,A -85,B 0,C 180,E1 -4728.696,E2 -4728.696} C_VEL
LIN {X 0,Y 523.912,Z 133.221,A -85,B 0,C 180,E1 -4731.898,E2 -4731.898} C_VEL
LIN {X 0,Y 523.917,Z 133.224,A -85,B 0,C 180,E1 -4734.913,E2 -4734.913} C_VEL
LIN {X 0,Y 523.936,Z 133.218,A -85,B 0,C 180,E1 -4737.68,E2 -4737.68} C_VEL
LIN {X 0,Y 523.938,Z 133.223,A -85,B 0,C 180,E1 -4740.681,E2 -4740.681} C_VEL
LIN {X 0,Y 523.904,Z 133.225,A -85,B 0,C 180,E1 -4743.725,E2 -4743.725} C_VEL
LIN {X 0,Y 523.935,Z 133.262,A -85,B 0,C 180,E1 -4745.537,E2 -4745.537} C_VEL
LIN {X 0,Y 525.346,Z 141.902,A -85,B 0,C 180,E1 -4746.964,E2 -4746.964} C_VEL
LIN {X 0,Y 524.9,Z 160.379,A -85,B 0,C 180,E1 -4749.832,E2 -4749.832} C_VEL
LIN {X 0,Y 524.532,Z 177.492,A -85,B 0,C 180,E1 -4752.454,E2 -4752.454} C_VEL
LIN {X 0,Y 524.21,Z 193.176,A -85,B 0,C 180,E1 -4754.833,E2 -4754.833} C_VEL
LIN {X 0,Y 525.884,Z 205.124,A -85,B 0,C 180,E1 -4755.055,E2 -4755.055} C_VEL
LIN {X 0,Y 525.494,Z 301.317,A -85,B 0,C 180,E1 -4756.391,E2 -4756.391} C_VEL
LIN {X 0,Y 525.291,Z 314.713,A -85,B 0,C 180,E1 -4756.73,E2 -4756.73} C_VEL
LIN {X 0,Y 525.01,Z 326.943,A -85,B 0,C 180,E1 -4757.19,E2 -4757.19} C_VEL
LIN {X 0,Y 524.738,Z 339.373,A -85,B 0,C 180,E1 -4757.828,E2 -4757.828} C_VEL
LIN {X 0,Y 524.478,Z 350.924,A -85,B 0,C 180,E1 -4758.601,E2 -4758.601} C_VEL
LIN {X 0,Y 524.202,Z 361.404,A -85,B 0,C 180,E1 -4759.475,E2 -4759.475} C_VEL
LIN {X 0,Y 523.948,Z 369.972,A -85,B 0,C 180,E1 -4760.348,E2 -4760.348} C_VEL
LIN {X 0,Y 523.761,Z 377.88,A -85,B 0,C 180,E1 -4761.318,E2 -4761.318} C_VEL
LIN {X 0,Y 523.595,Z 385.604,A -85,B 0,C 180,E1 -4762.48,E2 -4762.48} C_VEL
LIN {X 0,Y 523.46,Z 392.723,A -85,B 0,C 180,E1 -4763.834,E2 -4763.834} C_VEL
LIN {X 0,Y 523.383,Z 397.46,A -85,B 0,C 180,E1 -4764.993,E2 -4764.993} C_VEL
LIN {X 0,Y 523.443,Z 401.083,A -85,B 0,C 180,E1 -4766.151,E2 -4766.151} C_VEL
LIN {X 0,Y 523.368,Z 402.948,A -85,B 0,C 180,E1 -4766.921,E2 -4766.921} C_VEL
LIN {X 0,Y 523.335,Z 404.348,A -85,B 0,C 180,E1 -4767.691,E2 -4767.691} C_VEL
LIN {X 0,Y 523.256,Z 405.956,A -85,B 0,C 180,E1 -4769.231,E2 -4769.231} C_VEL
LIN {X 0,Y 523.257,Z 406.174,A -85,B 0,C 180,E1 -4770,E2 -4770} C_VEL
LIN {X 0,Y 523.275,Z 405.352,A -85,B 0,C 180,E1 -4771.539,E2 -4771.539} C_VEL
LIN {X 0,Y 523.335,Z 404.359,A -85,B 0,C 180,E1 -4772.309,E2 -4772.309} C_VEL
LIN {X 0,Y 523.368,Z 402.962,A -85,B 0,C 180,E1 -4773.079,E2 -4773.079} C_VEL
LIN {X 0,Y 523.423,Z 400.024,A -85,B 0,C 180,E1 -4774.235,E2 -4774.235} C_VEL
LIN {X 0,Y 523.456,Z 396.043,A -85,B 0,C 180,E1 -4775.393,E2 -4775.393} C_VEL
LIN {X 0,Y 523.509,Z 389.969,A -85,B 0,C 180,E1 -4776.737,E2 -4776.737} C_VEL
LIN {X 0,Y 523.645,Z 383.229,A -85,B 0,C 180,E1 -4777.907,E2 -4777.907} C_VEL
LIN {X 0,Y 523.827,Z 374.928,A -85,B 0,C 180,E1 -4779.07,E2 -4779.07} C_VEL
LIN {X 0,Y 524.03,Z 366.417,A -85,B 0,C 180,E1 -4780.041,E2 -4780.041} C_VEL
LIN {X 0,Y 524.309,Z 355.902,A -85,B 0,C 180,E1 -4781.012,E2 -4781.012} C_VEL
LIN {X 0,Y 524.596,Z 345.687,A -85,B 0,C 180,E1 -4781.776,E2 -4781.776} C_VEL
LIN {X 0,Y 524.888,Z 334.097,A -85,B 0,C 180,E1 -4782.469,E2 -4782.469} C_VEL
LIN {X 0,Y 525.109,Z 322.372,A -85,B 0,C 180,E1 -4783.004,E2 -4783.004} C_VEL
LIN {X 0,Y 525.359,Z 308.864,A -85,B 0,C 180,E1 -4783.441,E2 -4783.441} C_VEL
LIN {X 0,Y 525.55,Z 295.401,A -85,B 0,C 180,E1 -4783.707,E2 -4783.707} C_VEL
